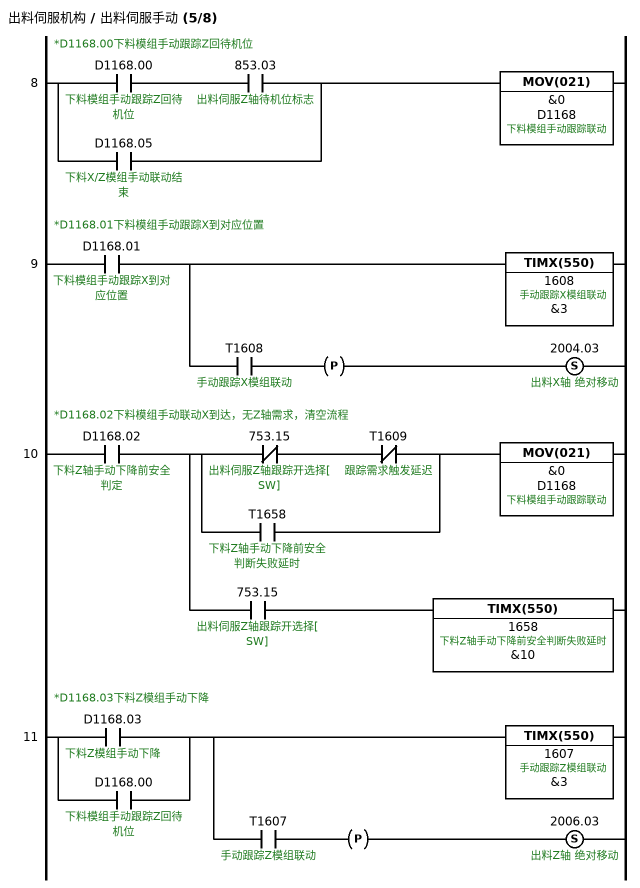
; [picture p480: 出料伺服机构 / 出料伺服手动, rungs 8-11]
; rung 8: *D1168.00下料模组手动跟踪Z回待机位
LD D1168.00  ; 下料模组手动跟踪Z回待机位
AND 853.03  ; 出料伺服Z轴待机位标志
OR D1168.05  ; 下料X/Z模组手动联动结束
MOV(021) &0 D1168  ; 下料模组手动跟踪联动
; rung 9: *D1168.01下料模组手动跟踪X到对应位置
LD D1168.01  ; 下料模组手动跟踪X到对应位置
TIMX(550) 1608 &3  ; 手动跟踪X模组联动
AND T1608  ; 手动跟踪X模组联动
UP(521)
SET 2004.03  ; 出料X轴 绝对移动
; rung 10: *D1168.02下料模组手动联动X到达，无Z轴需求，清空流程
LD D1168.02  ; 下料Z轴手动下降前安全判定
OUT TR0
LDNOT 753.15  ; 出料伺服Z轴跟踪开选择[SW]
ANDNOT T1609  ; 跟踪需求触发延迟
OR T1658  ; 下料Z轴手动下降前安全判断失败延时
ANDLD
MOV(021) &0 D1168  ; 下料模组手动跟踪联动
LD TR0
AND 753.15  ; 出料伺服Z轴跟踪开选择[SW]
TIMX(550) 1658 &10  ; 下料Z轴手动下降前安全判断失败延时
; rung 11: *D1168.03下料Z模组手动下降
LD D1168.03  ; 下料Z模组手动下降
OR D1168.00  ; 下料模组手动跟踪Z回待机位
TIMX(550) 1607 &3  ; 手动跟踪Z模组联动
AND T1607  ; 手动跟踪Z模组联动
UP(521)
SET 2006.03  ; 出料Z轴 绝对移动

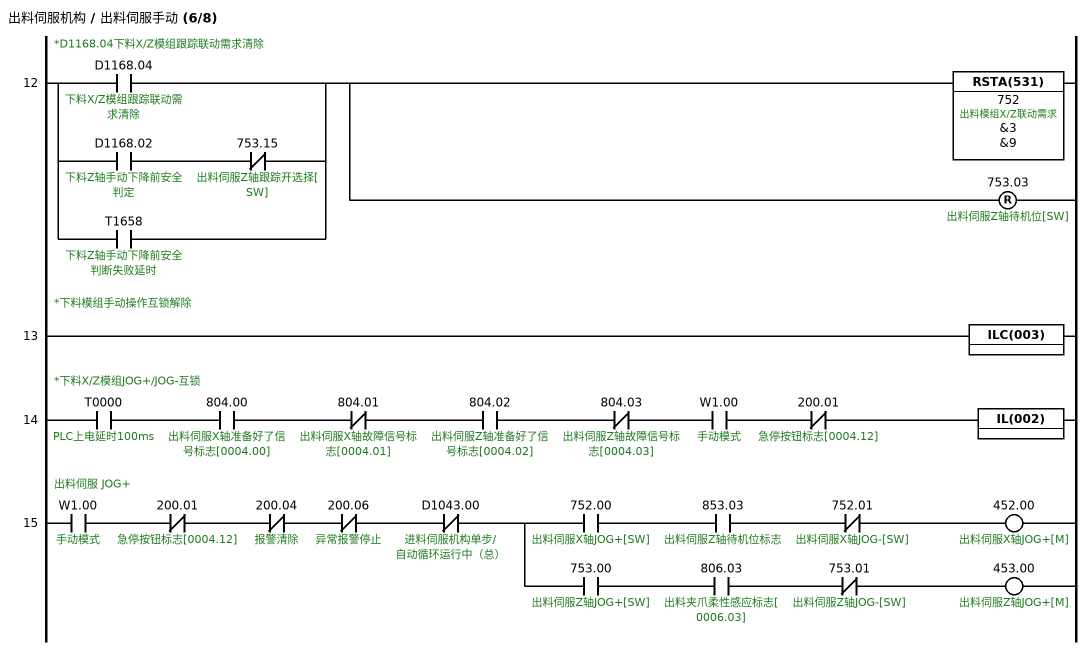
; rung 12: *D1168.04下料X/Z模组跟踪联动需求清除
LD D1168.04  ; 下料X/Z模组跟踪联动需求清除
LD D1168.02  ; 下料Z轴手动下降前安全判定
ANDNOT 753.15  ; 出料伺服Z轴跟踪开选择[SW]
ORLD
OR T1658  ; 下料Z轴手动下降前安全判断失败延时
RSTA(531) 752 &3 &9  ; 出料模组X/Z联动需求
RSET 753.03  ; 出料伺服Z轴待机位[SW]
; rung 13: *下料模组手动操作互锁解除
ILC(003)
; rung 14: *下料X/Z模组JOG+/JOG-互锁
LD T0000  ; PLC上电延时100ms
AND 804.00  ; 出料伺服X轴准备好了信号标志[0004.00]
ANDNOT 804.01  ; 出料伺服X轴故障信号标志[0004.01]
AND 804.02  ; 出料伺服Z轴准备好了信号标志[0004.02]
ANDNOT 804.03  ; 出料伺服Z轴故障信号标志[0004.03]
AND W1.00  ; 手动模式
ANDNOT 200.01  ; 急停按钮标志[0004.12]
IL(002)
; rung 15: 出料伺服 JOG+
LD W1.00  ; 手动模式
ANDNOT 200.01  ; 急停按钮标志[0004.12]
ANDNOT 200.04  ; 报警清除
ANDNOT 200.06  ; 异常报警停止
ANDNOT D1043.00  ; 进料伺服机构单步/自动循环运行中（总）
OUT TR0
AND 752.00  ; 出料伺服X轴JOG+[SW]
AND 853.03  ; 出料伺服Z轴待机位标志
ANDNOT 752.01  ; 出料伺服X轴JOG-[SW]
OUT 452.00  ; 出料伺服X轴JOG+[M]
LD TR0
AND 753.00  ; 出料伺服Z轴JOG+[SW]
AND 806.03  ; 出料夹爪柔性感应标志[0006.03]
ANDNOT 753.01  ; 出料伺服Z轴JOG-[SW]
OUT 453.00  ; 出料伺服Z轴JOG+[M]

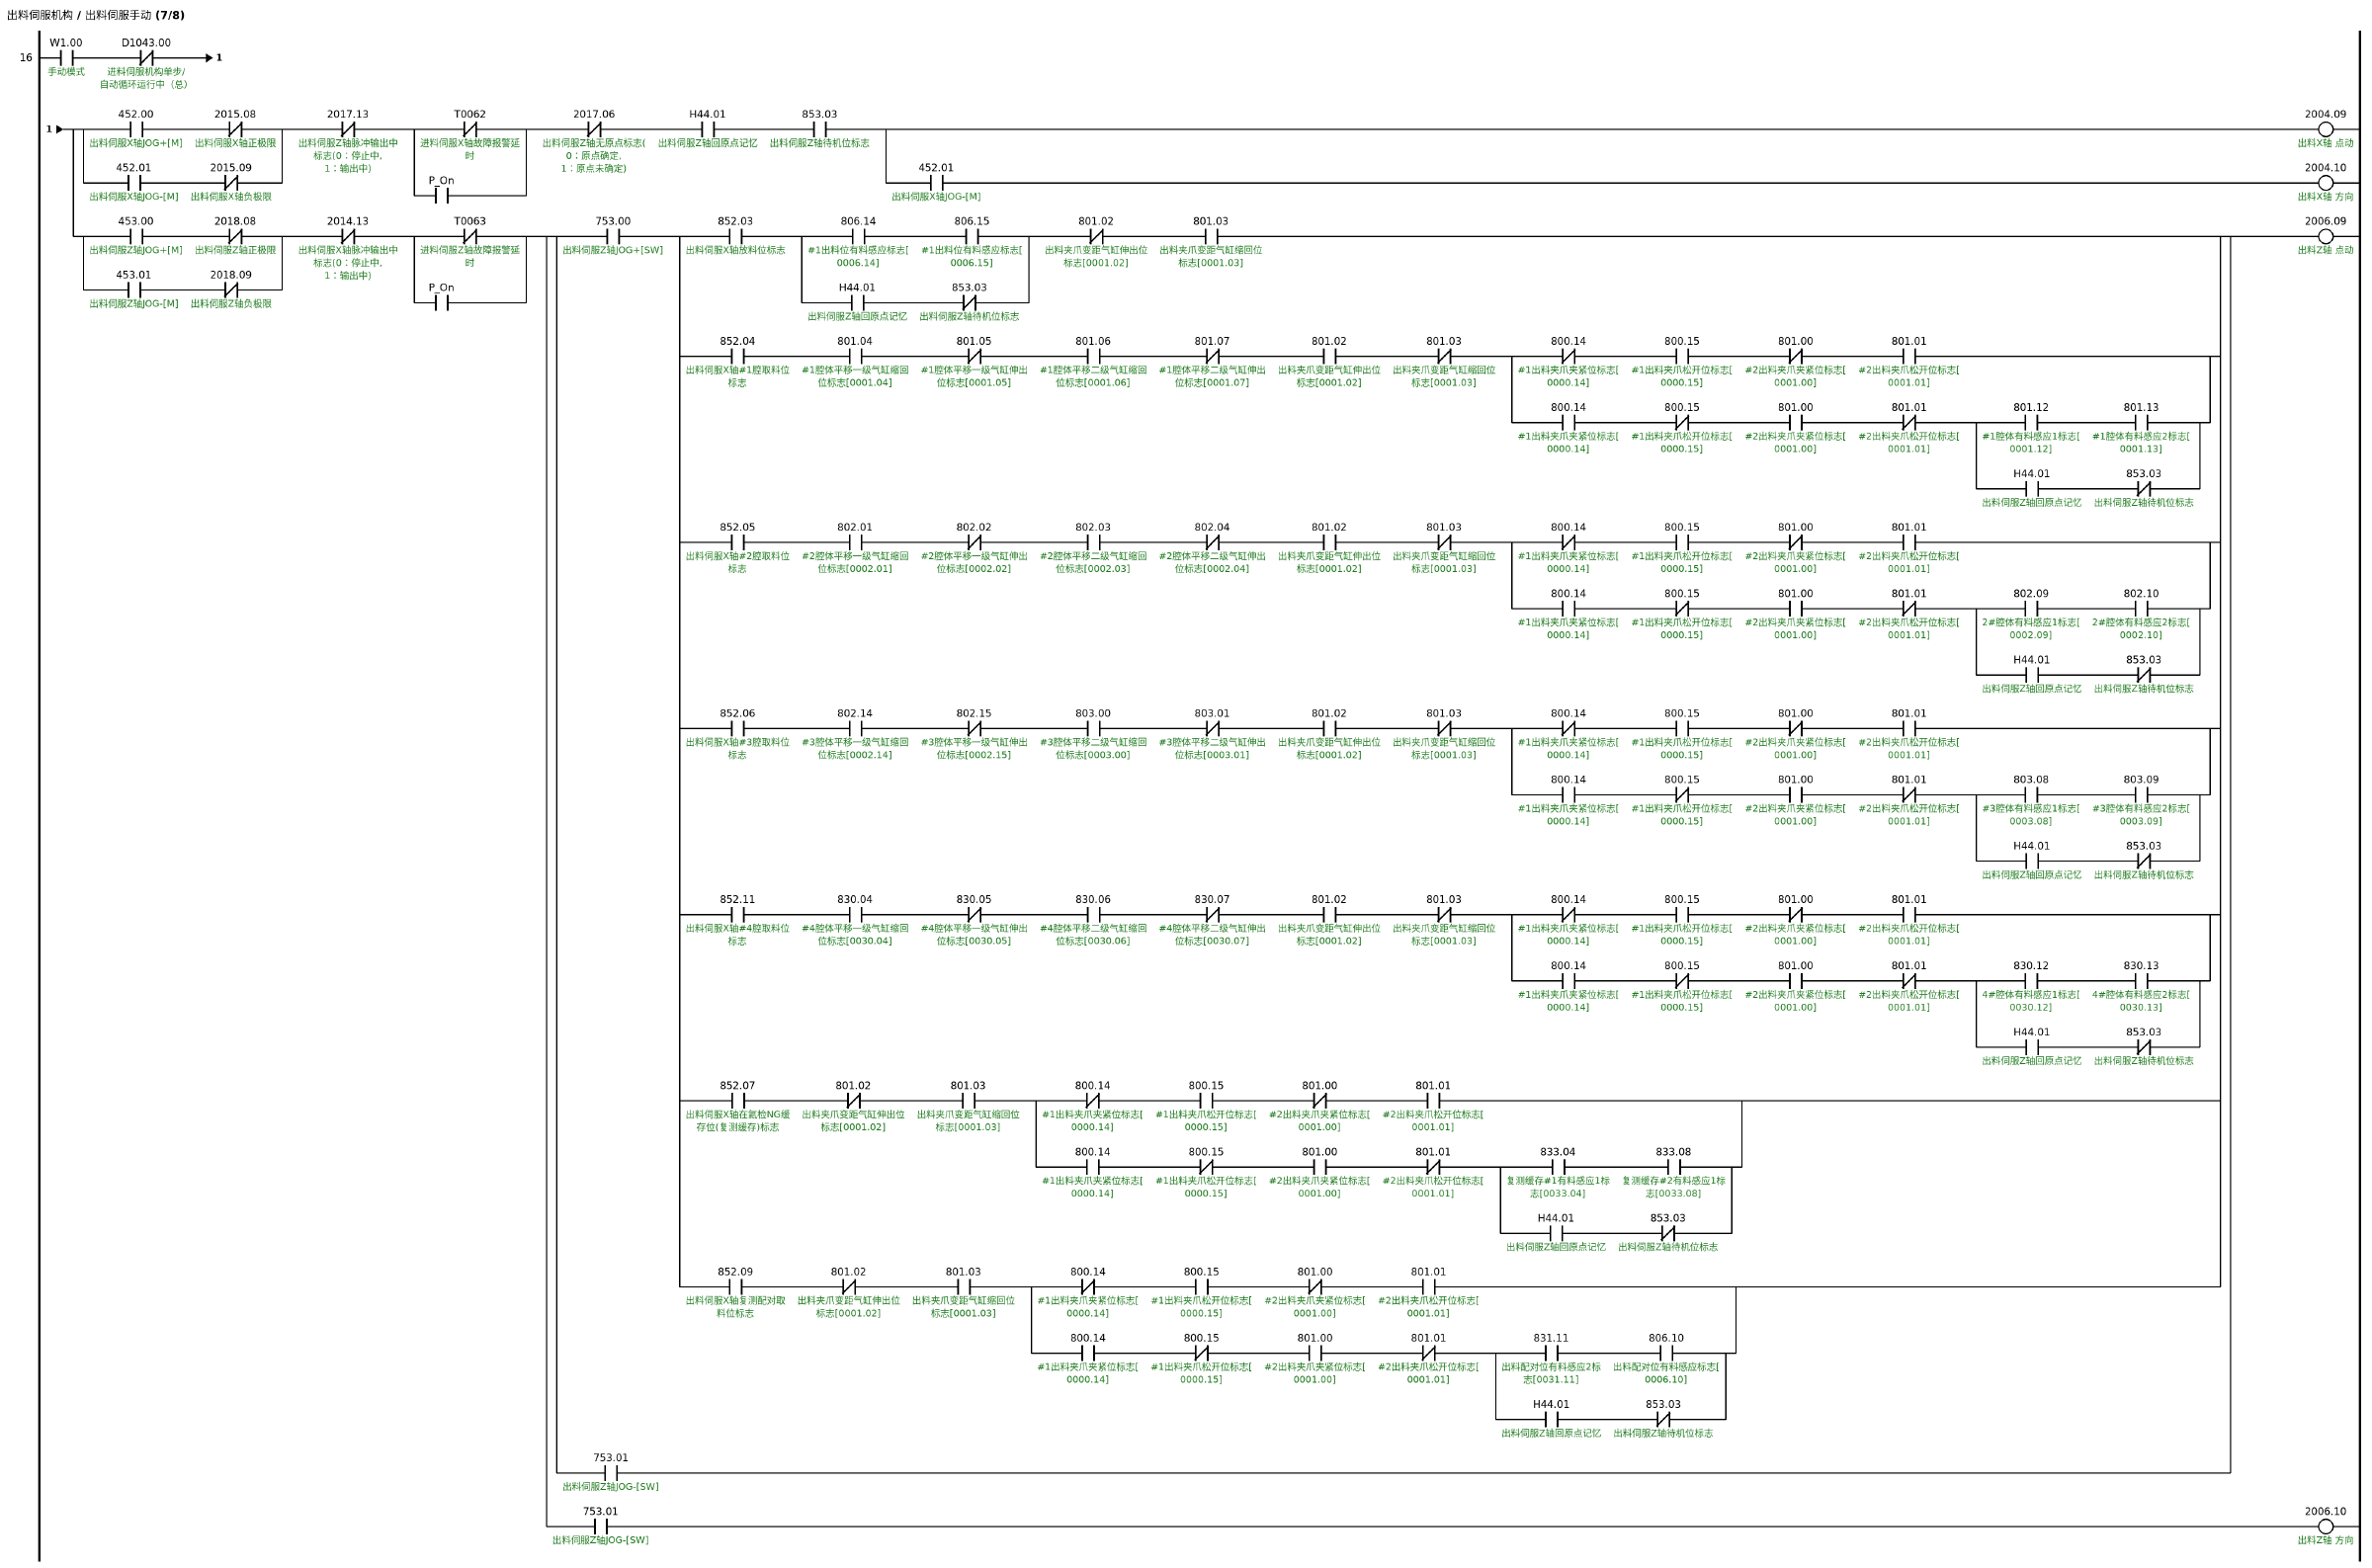
; rung 16
LD W1.00  ; 手动模式
ANDNOT D1043.00  ; 进料伺服机构单步/自动循环运行中（总）
OUT TR0
LD 452.00  ; 出料伺服X轴JOG+[M]
ANDNOT 2015.08  ; 出料伺服X轴正极限
LD 452.01  ; 出料伺服X轴JOG-[M]
ANDNOT 2015.09  ; 出料伺服X轴负极限
ORLD
ANDLD
ANDNOT 2017.13  ; 出料伺服Z轴脉冲输出中标志(0：停止中,1：输出中)
LDNOT T0062  ; 进料伺服X轴故障报警延时
OR P_On
ANDLD
ANDNOT 2017.06  ; 出料伺服Z轴无原点标志(0：原点确定,1：原点未确定)
AND H44.01  ; 出料伺服Z轴回原点记忆
AND 853.03  ; 出料伺服Z轴待机位标志
OUT 2004.09  ; 出料X轴 点动
AND 452.01  ; 出料伺服X轴JOG-[M]
OUT 2004.10  ; 出料X轴 方向
LD TR0
LD 453.00  ; 出料伺服Z轴JOG+[M]
ANDNOT 2018.08  ; 出料伺服Z轴正极限
LD 453.01  ; 出料伺服Z轴JOG-[M]
ANDNOT 2018.09  ; 出料伺服Z轴负极限
ORLD
ANDLD
ANDNOT 2014.13  ; 出料伺服X轴脉冲输出中标志(0：停止中,1：输出中)
LDNOT T0063  ; 进料伺服Z轴故障报警延时
OR P_On
ANDLD
OUT TR0
LD 753.00  ; 出料伺服Z轴JOG+[SW]
LD 852.03  ; 出料伺服X轴放料位标志
LD 806.14  ; #1出料位有料感应标志[0006.14]
AND 806.15  ; #1出料位有料感应标志[0006.15]
LD H44.01  ; 出料伺服Z轴回原点记忆
ANDNOT 853.03  ; 出料伺服Z轴待机位标志
ORLD
ANDLD
ANDNOT 801.02  ; 出料夹爪变距气缸伸出位标志[0001.02]
AND 801.03  ; 出料夹爪变距气缸缩回位标志[0001.03]
LD 852.04  ; 出料伺服X轴#1腔取料位标志
AND 801.04  ; #1腔体平移一级气缸缩回位标志[0001.04]
ANDNOT 801.05  ; #1腔体平移一级气缸伸出位标志[0001.05]
AND 801.06  ; #1腔体平移二级气缸缩回位标志[0001.06]
ANDNOT 801.07  ; #1腔体平移二级气缸伸出位标志[0001.07]
AND 801.02  ; 出料夹爪变距气缸伸出位标志[0001.02]
ANDNOT 801.03  ; 出料夹爪变距气缸缩回位标志[0001.03]
LDNOT 800.14  ; #1出料夹爪夹紧位标志[0000.14]
AND 800.15  ; #1出料夹爪松开位标志[0000.15]
ANDNOT 801.00  ; #2出料夹爪夹紧位标志[0001.00]
AND 801.01  ; #2出料夹爪松开位标志[0001.01]
LD 800.14  ; #1出料夹爪夹紧位标志[0000.14]
ANDNOT 800.15  ; #1出料夹爪松开位标志[0000.15]
AND 801.00  ; #2出料夹爪夹紧位标志[0001.00]
ANDNOT 801.01  ; #2出料夹爪松开位标志[0001.01]
LD 801.12  ; #1腔体有料感应1标志[0001.12]
AND 801.13  ; #1腔体有料感应2标志[0001.13]
LD H44.01  ; 出料伺服Z轴回原点记忆
ANDNOT 853.03  ; 出料伺服Z轴待机位标志
ORLD
ANDLD
ORLD
ANDLD
ORLD
LD 852.05  ; 出料伺服X轴#2腔取料位标志
AND 802.01  ; #2腔体平移一级气缸缩回位标志[0002.01]
ANDNOT 802.02  ; #2腔体平移一级气缸伸出位标志[0002.02]
AND 802.03  ; #2腔体平移二级气缸缩回位标志[0002.03]
ANDNOT 802.04  ; #2腔体平移二级气缸伸出位标志[0002.04]
AND 801.02  ; 出料夹爪变距气缸伸出位标志[0001.02]
ANDNOT 801.03  ; 出料夹爪变距气缸缩回位标志[0001.03]
LDNOT 800.14  ; #1出料夹爪夹紧位标志[0000.14]
AND 800.15  ; #1出料夹爪松开位标志[0000.15]
ANDNOT 801.00  ; #2出料夹爪夹紧位标志[0001.00]
AND 801.01  ; #2出料夹爪松开位标志[0001.01]
LD 800.14  ; #1出料夹爪夹紧位标志[0000.14]
ANDNOT 800.15  ; #1出料夹爪松开位标志[0000.15]
AND 801.00  ; #2出料夹爪夹紧位标志[0001.00]
ANDNOT 801.01  ; #2出料夹爪松开位标志[0001.01]
LD 802.09  ; 2#腔体有料感应1标志[0002.09]
AND 802.10  ; 2#腔体有料感应2标志[0002.10]
LD H44.01  ; 出料伺服Z轴回原点记忆
ANDNOT 853.03  ; 出料伺服Z轴待机位标志
ORLD
ANDLD
ORLD
ANDLD
ORLD
LD 852.06  ; 出料伺服X轴#3腔取料位标志
AND 802.14  ; #3腔体平移一级气缸缩回位标志[0002.14]
ANDNOT 802.15  ; #3腔体平移一级气缸伸出位标志[0002.15]
AND 803.00  ; #3腔体平移二级气缸缩回位标志[0003.00]
ANDNOT 803.01  ; #3腔体平移二级气缸伸出位标志[0003.01]
AND 801.02  ; 出料夹爪变距气缸伸出位标志[0001.02]
ANDNOT 801.03  ; 出料夹爪变距气缸缩回位标志[0001.03]
LDNOT 800.14  ; #1出料夹爪夹紧位标志[0000.14]
AND 800.15  ; #1出料夹爪松开位标志[0000.15]
ANDNOT 801.00  ; #2出料夹爪夹紧位标志[0001.00]
AND 801.01  ; #2出料夹爪松开位标志[0001.01]
LD 800.14  ; #1出料夹爪夹紧位标志[0000.14]
ANDNOT 800.15  ; #1出料夹爪松开位标志[0000.15]
AND 801.00  ; #2出料夹爪夹紧位标志[0001.00]
ANDNOT 801.01  ; #2出料夹爪松开位标志[0001.01]
LD 803.08  ; #3腔体有料感应1标志[0003.08]
AND 803.09  ; #3腔体有料感应2标志[0003.09]
LD H44.01  ; 出料伺服Z轴回原点记忆
ANDNOT 853.03  ; 出料伺服Z轴待机位标志
ORLD
ANDLD
ORLD
ANDLD
ORLD
LD 852.11  ; 出料伺服X轴#4腔取料位标志
AND 830.04  ; #4腔体平移一级气缸缩回位标志[0030.04]
ANDNOT 830.05  ; #4腔体平移一级气缸伸出位标志[0030.05]
AND 830.06  ; #4腔体平移二级气缸缩回位标志[0030.06]
ANDNOT 830.07  ; #4腔体平移二级气缸伸出位标志[0030.07]
AND 801.02  ; 出料夹爪变距气缸伸出位标志[0001.02]
ANDNOT 801.03  ; 出料夹爪变距气缸缩回位标志[0001.03]
LDNOT 800.14  ; #1出料夹爪夹紧位标志[0000.14]
AND 800.15  ; #1出料夹爪松开位标志[0000.15]
ANDNOT 801.00  ; #2出料夹爪夹紧位标志[0001.00]
AND 801.01  ; #2出料夹爪松开位标志[0001.01]
LD 800.14  ; #1出料夹爪夹紧位标志[0000.14]
ANDNOT 800.15  ; #1出料夹爪松开位标志[0000.15]
AND 801.00  ; #2出料夹爪夹紧位标志[0001.00]
ANDNOT 801.01  ; #2出料夹爪松开位标志[0001.01]
LD 830.12  ; 4#腔体有料感应1标志[0030.12]
AND 830.13  ; 4#腔体有料感应2标志[0030.13]
LD H44.01  ; 出料伺服Z轴回原点记忆
ANDNOT 853.03  ; 出料伺服Z轴待机位标志
ORLD
ANDLD
ORLD
ANDLD
ORLD
LD 852.07  ; 出料伺服X轴在氦检NG缓存位(复测缓存)标志
ANDNOT 801.02  ; 出料夹爪变距气缸伸出位标志[0001.02]
AND 801.03  ; 出料夹爪变距气缸缩回位标志[0001.03]
LDNOT 800.14  ; #1出料夹爪夹紧位标志[0000.14]
AND 800.15  ; #1出料夹爪松开位标志[0000.15]
ANDNOT 801.00  ; #2出料夹爪夹紧位标志[0001.00]
AND 801.01  ; #2出料夹爪松开位标志[0001.01]
LD 800.14  ; #1出料夹爪夹紧位标志[0000.14]
ANDNOT 800.15  ; #1出料夹爪松开位标志[0000.15]
AND 801.00  ; #2出料夹爪夹紧位标志[0001.00]
ANDNOT 801.01  ; #2出料夹爪松开位标志[0001.01]
LD 833.04  ; 复测缓存#1有料感应1标志[0033.04]
AND 833.08  ; 复测缓存#2有料感应1标志[0033.08]
LD H44.01  ; 出料伺服Z轴回原点记忆
ANDNOT 853.03  ; 出料伺服Z轴待机位标志
ORLD
ANDLD
ORLD
ANDLD
ORLD
LD 852.09  ; 出料伺服X轴复测配对取料位标志
ANDNOT 801.02  ; 出料夹爪变距气缸伸出位标志[0001.02]
AND 801.03  ; 出料夹爪变距气缸缩回位标志[0001.03]
LDNOT 800.14  ; #1出料夹爪夹紧位标志[0000.14]
AND 800.15  ; #1出料夹爪松开位标志[0000.15]
ANDNOT 801.00  ; #2出料夹爪夹紧位标志[0001.00]
AND 801.01  ; #2出料夹爪松开位标志[0001.01]
LD 800.14  ; #1出料夹爪夹紧位标志[0000.14]
ANDNOT 800.15  ; #1出料夹爪松开位标志[0000.15]
AND 801.00  ; #2出料夹爪夹紧位标志[0001.00]
ANDNOT 801.01  ; #2出料夹爪松开位标志[0001.01]
LD 831.11  ; 出料配对位有料感应2标志[0031.11]
AND 806.10  ; 出料配对位有料感应标志[0006.10]
LD H44.01  ; 出料伺服Z轴回原点记忆
ANDNOT 853.03  ; 出料伺服Z轴待机位标志
ORLD
ANDLD
ORLD
ANDLD
ORLD
ANDLD
OR 753.01  ; 出料伺服Z轴JOG-[SW]
ANDLD
OUT 2006.09  ; 出料Z轴 点动
LD TR0
AND 753.01  ; 出料伺服Z轴JOG-[SW]
OUT 2006.10  ; 出料Z轴 方向

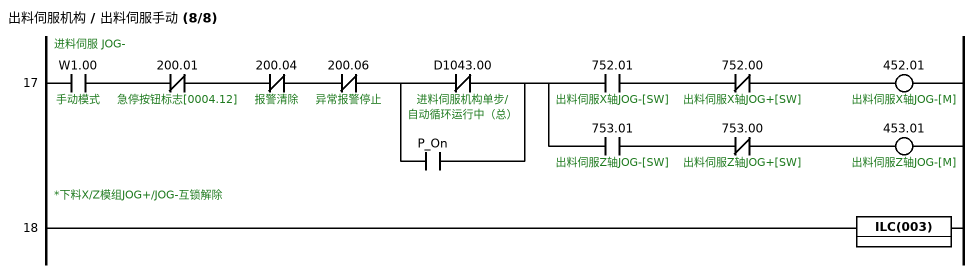
; rung 17: 进料伺服 JOG-
LD W1.00  ; 手动模式
ANDNOT 200.01  ; 急停按钮标志[0004.12]
ANDNOT 200.04  ; 报警清除
ANDNOT 200.06  ; 异常报警停止
LDNOT D1043.00  ; 进料伺服机构单步/自动循环运行中（总）
OR P_On
ANDLD
OUT TR0
AND 752.01  ; 出料伺服X轴JOG-[SW]
ANDNOT 752.00  ; 出料伺服X轴JOG+[SW]
OUT 452.01  ; 出料伺服X轴JOG-[M]
LD TR0
AND 753.01  ; 出料伺服Z轴JOG-[SW]
ANDNOT 753.00  ; 出料伺服Z轴JOG+[SW]
OUT 453.01  ; 出料伺服Z轴JOG-[M]
; rung 18: *下料X/Z模组JOG+/JOG-互锁解除
ILC(003)

### Section 出料伺服自动

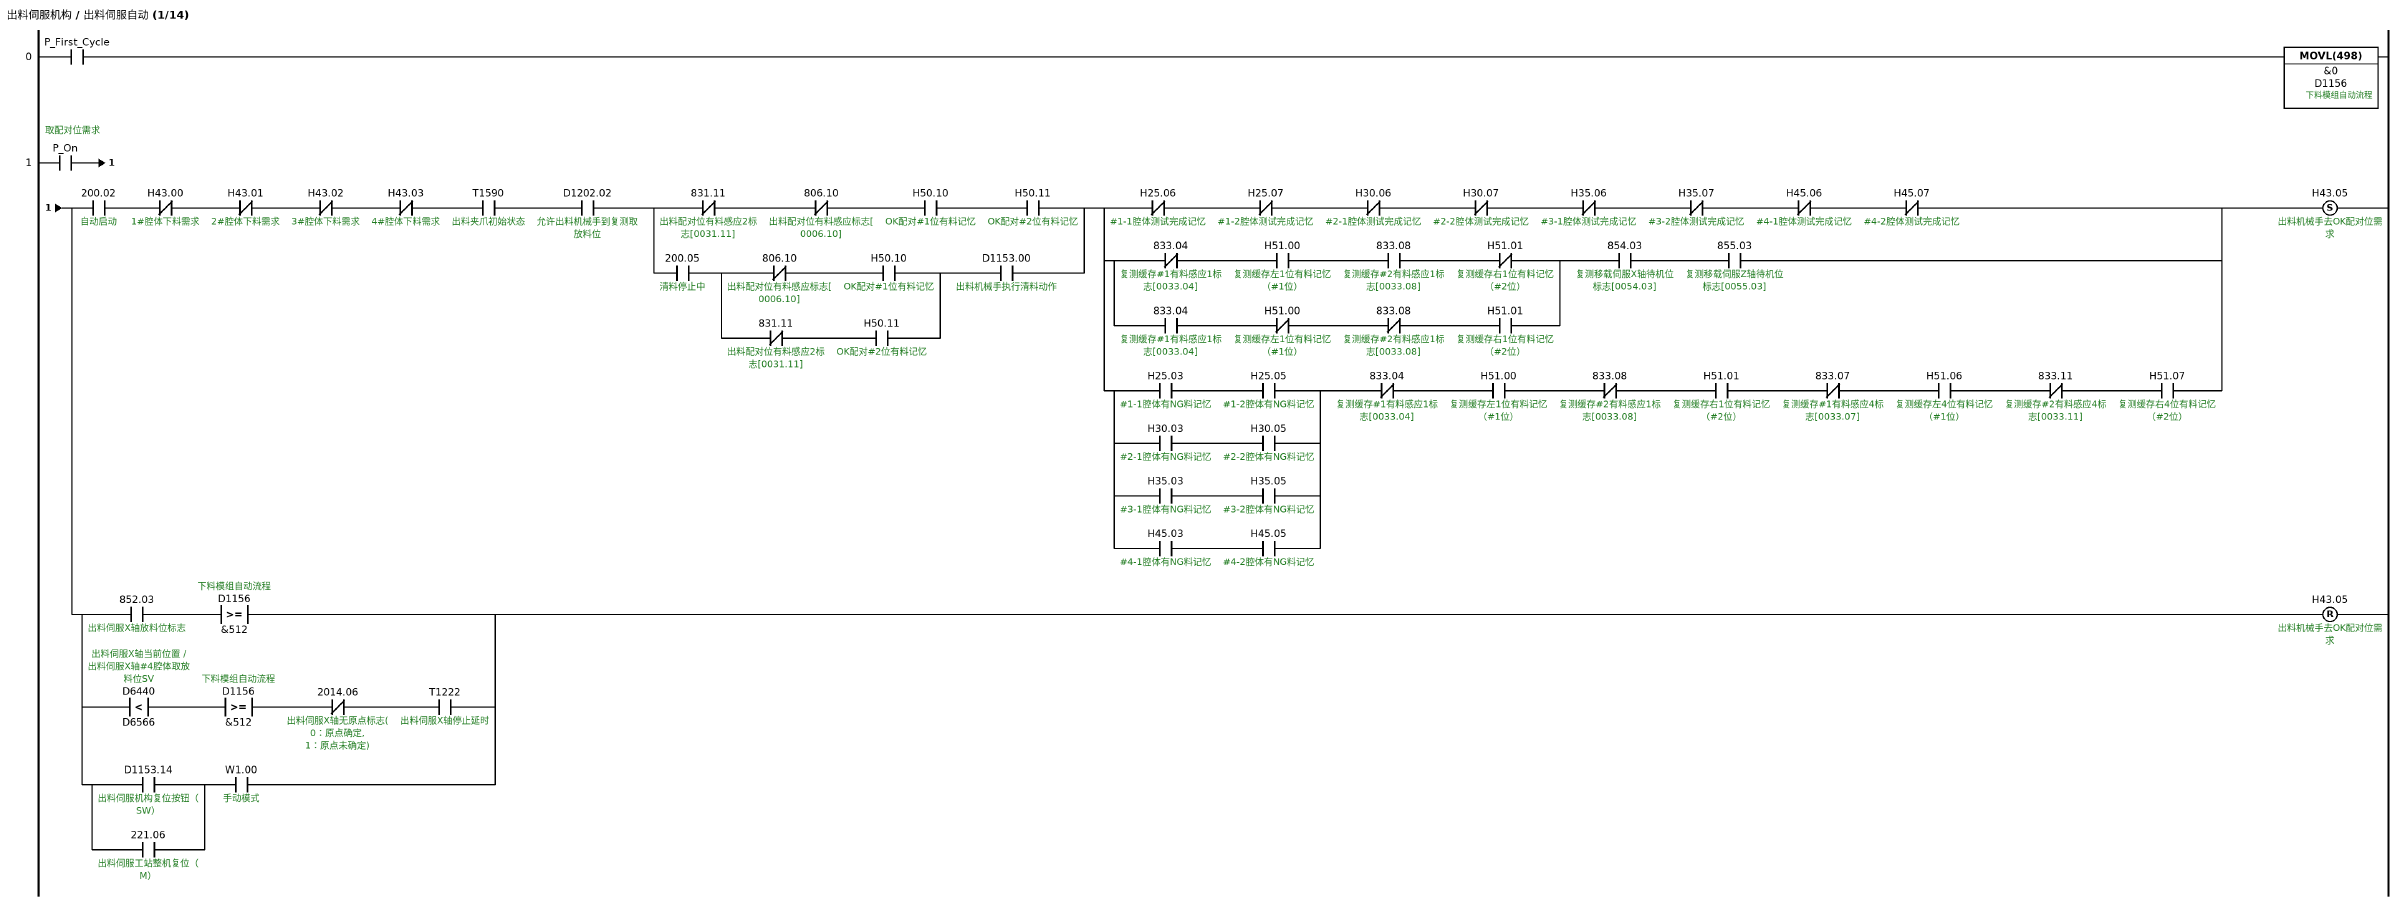
; rung 0
LD P_First_Cycle
MOVL(498) &0 D1156  ; 下料模组自动流程
; rung 1: 取配对位需求
LD P_On
OUT TR0
AND 200.02  ; 自动启动
ANDNOT H43.00  ; 1#腔体下料需求
ANDNOT H43.01  ; 2#腔体下料需求
ANDNOT H43.02  ; 3#腔体下料需求
ANDNOT H43.03  ; 4#腔体下料需求
AND T1590  ; 出料夹爪初始状态
AND D1202.02  ; 允许出料机械手到复测取放料位
LDNOT 831.11  ; 出料配对位有料感应2标志[0031.11]
ANDNOT 806.10  ; 出料配对位有料感应标志[0006.10]
AND H50.10  ; OK配对#1位有料记忆
AND H50.11  ; OK配对#2位有料记忆
LD 200.05  ; 清料停止中
LDNOT 806.10  ; 出料配对位有料感应标志[0006.10]
AND H50.10  ; OK配对#1位有料记忆
LDNOT 831.11  ; 出料配对位有料感应2标志[0031.11]
AND H50.11  ; OK配对#2位有料记忆
ORLD
ANDLD
AND D1153.00  ; 出料机械手执行清料动作
ORLD
ANDLD
LDNOT H25.06  ; #1-1腔体测试完成记忆
ANDNOT H25.07  ; #1-2腔体测试完成记忆
ANDNOT H30.06  ; #2-1腔体测试完成记忆
ANDNOT H30.07  ; #2-2腔体测试完成记忆
ANDNOT H35.06  ; #3-1腔体测试完成记忆
ANDNOT H35.07  ; #3-2腔体测试完成记忆
ANDNOT H45.06  ; #4-1腔体测试完成记忆
ANDNOT H45.07  ; #4-2腔体测试完成记忆
LDNOT 833.04  ; 复测缓存#1有料感应1标志[0033.04]
AND H51.00  ; 复测缓存左1位有料记忆（#1位）
AND 833.08  ; 复测缓存#2有料感应1标志[0033.08]
ANDNOT H51.01  ; 复测缓存右1位有料记忆（#2位）
LD 833.04  ; 复测缓存#1有料感应1标志[0033.04]
ANDNOT H51.00  ; 复测缓存左1位有料记忆（#1位）
ANDNOT 833.08  ; 复测缓存#2有料感应1标志[0033.08]
AND H51.01  ; 复测缓存右1位有料记忆（#2位）
ORLD
AND 854.03  ; 复测移载伺服X轴待机位标志[0054.03]
AND 855.03  ; 复测移载伺服Z轴待机位标志[0055.03]
ORLD
LD H25.03  ; #1-1腔体有NG料记忆
AND H25.05  ; #1-2腔体有NG料记忆
LD H30.03  ; #2-1腔体有NG料记忆
AND H30.05  ; #2-2腔体有NG料记忆
ORLD
LD H35.03  ; #3-1腔体有NG料记忆
AND H35.05  ; #3-2腔体有NG料记忆
ORLD
LD H45.03  ; #4-1腔体有NG料记忆
AND H45.05  ; #4-2腔体有NG料记忆
ORLD
ANDNOT 833.04  ; 复测缓存#1有料感应1标志[0033.04]
AND H51.00  ; 复测缓存左1位有料记忆（#1位）
ANDNOT 833.08  ; 复测缓存#2有料感应1标志[0033.08]
AND H51.01  ; 复测缓存右1位有料记忆（#2位）
ANDNOT 833.07  ; 复测缓存#1有料感应4标志[0033.07]
AND H51.06  ; 复测缓存左4位有料记忆（#1位）
ANDNOT 833.11  ; 复测缓存#2有料感应4标志[0033.11]
AND H51.07  ; 复测缓存右4位有料记忆（#2位）
ORLD
ANDLD
SET H43.05  ; 出料机械手去OK配对位需求
LD TR0
LD 852.03  ; 出料伺服X轴放料位标志
AND>=(325) D1156 &512  ; 下料模组自动流程
LD<SL(313) D6440 D6566  ; 出料伺服X轴当前位置, 出料伺服X轴#4腔体取放料位SV
AND>=(325) D1156 &512  ; 下料模组自动流程
ANDNOT 2014.06  ; 出料伺服X轴无原点标志(0：原点确定,1：原点未确定)
AND T1222  ; 出料伺服X轴停止延时
ORLD
LD D1153.14  ; 出料伺服机构复位按钮（SW）
OR 221.06  ; 出料伺服工站整机复位（M）
AND W1.00  ; 手动模式
ORLD
ANDLD
RSET H43.05  ; 出料机械手去OK配对位需求

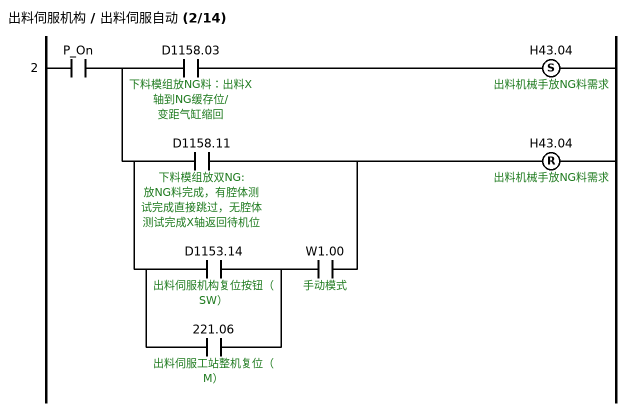
; rung 2
LD P_On
OUT TR0
AND D1158.03  ; 下料模组放NG料：出料X轴到NG缓存位/变距气缸缩回
SET H43.04  ; 出料机械手放NG料需求
LD TR0
LD D1158.11  ; 下料模组放双NG:放NG料完成，有腔体测试完成直接跳过，无腔体测试完成X轴返回待机位
LD D1153.14  ; 出料伺服机构复位按钮（SW）
OR 221.06  ; 出料伺服工站整机复位（M）
AND W1.00  ; 手动模式
ORLD
ANDLD
RSET H43.04  ; 出料机械手放NG料需求

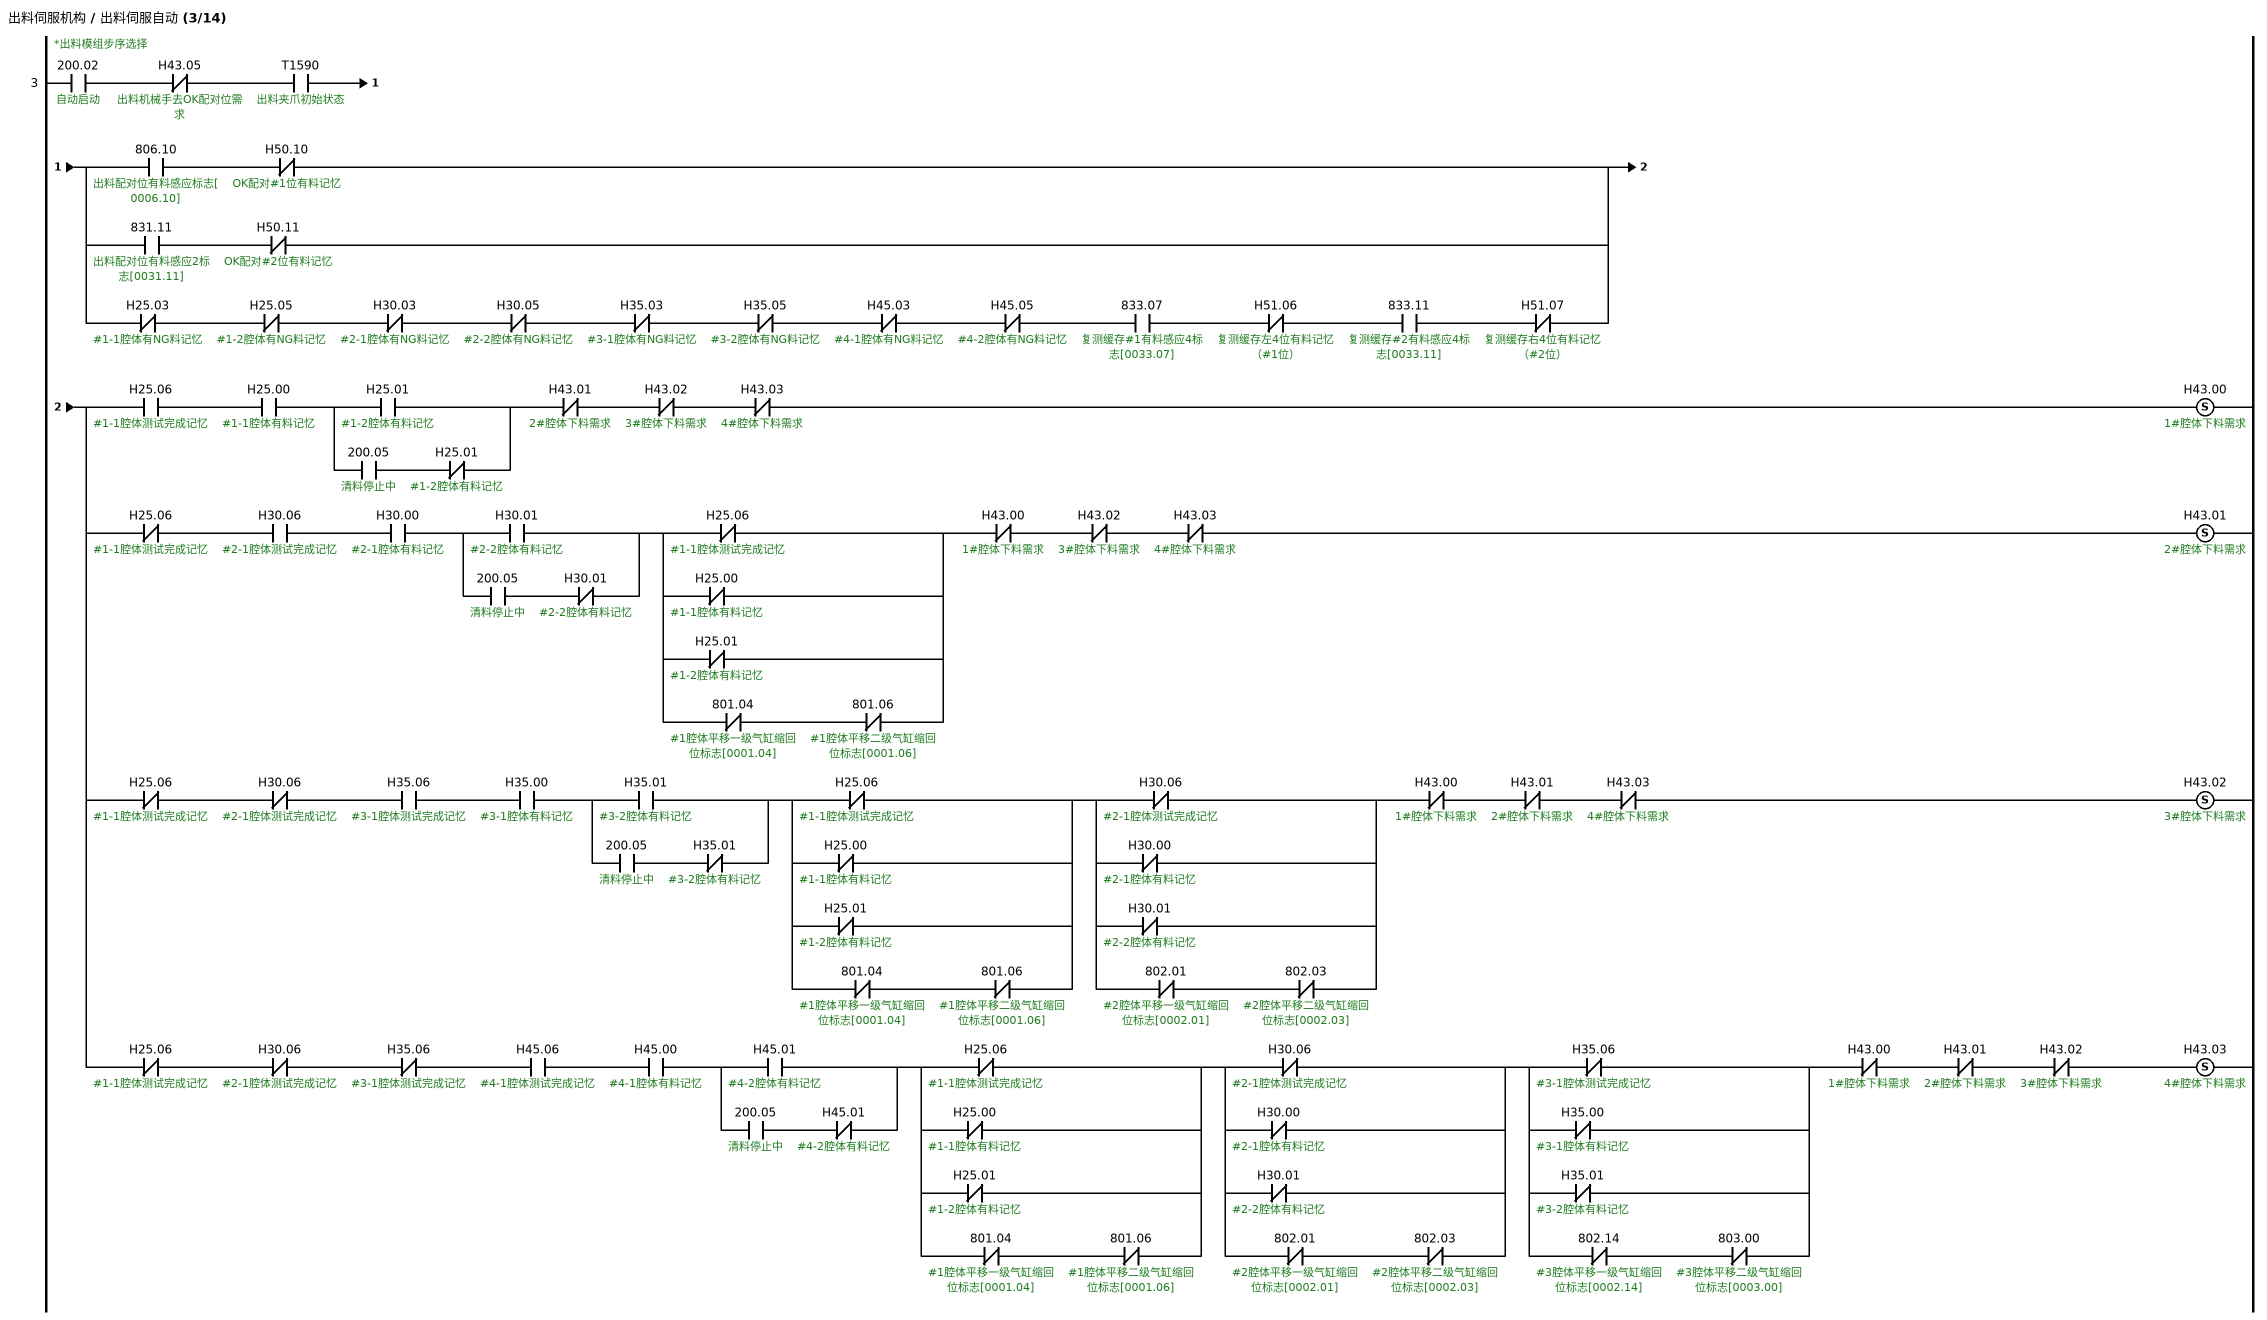
; rung 3: *出料模组步序选择
LD 200.02  ; 自动启动
ANDNOT H43.05  ; 出料机械手去OK配对位需求
AND T1590  ; 出料夹爪初始状态
LD 806.10  ; 出料配对位有料感应标志[0006.10]
ANDNOT H50.10  ; OK配对#1位有料记忆
LD 831.11  ; 出料配对位有料感应2标志[0031.11]
ANDNOT H50.11  ; OK配对#2位有料记忆
ORLD
LDNOT H25.03  ; #1-1腔体有NG料记忆
ANDNOT H25.05  ; #1-2腔体有NG料记忆
ANDNOT H30.03  ; #2-1腔体有NG料记忆
ANDNOT H30.05  ; #2-2腔体有NG料记忆
ANDNOT H35.03  ; #3-1腔体有NG料记忆
ANDNOT H35.05  ; #3-2腔体有NG料记忆
ANDNOT H45.03  ; #4-1腔体有NG料记忆
ANDNOT H45.05  ; #4-2腔体有NG料记忆
AND 833.07  ; 复测缓存#1有料感应4标志[0033.07]
ANDNOT H51.06  ; 复测缓存左4位有料记忆（#1位）
AND 833.11  ; 复测缓存#2有料感应4标志[0033.11]
ANDNOT H51.07  ; 复测缓存右4位有料记忆（#2位）
ORLD
ANDLD
OUT TR0
AND H25.06  ; #1-1腔体测试完成记忆
AND H25.00  ; #1-1腔体有料记忆
LD H25.01  ; #1-2腔体有料记忆
LD 200.05  ; 清料停止中
ANDNOT H25.01  ; #1-2腔体有料记忆
ORLD
ANDLD
ANDNOT H43.01  ; 2#腔体下料需求
ANDNOT H43.02  ; 3#腔体下料需求
ANDNOT H43.03  ; 4#腔体下料需求
SET H43.00  ; 1#腔体下料需求
LD TR0
ANDNOT H25.06  ; #1-1腔体测试完成记忆
AND H30.06  ; #2-1腔体测试完成记忆
AND H30.00  ; #2-1腔体有料记忆
LD H30.01  ; #2-2腔体有料记忆
LD 200.05  ; 清料停止中
ANDNOT H30.01  ; #2-2腔体有料记忆
ORLD
ANDLD
LDNOT H25.06  ; #1-1腔体测试完成记忆
ORNOT H25.00  ; #1-1腔体有料记忆
ORNOT H25.01  ; #1-2腔体有料记忆
LDNOT 801.04  ; #1腔体平移一级气缸缩回位标志[0001.04]
ANDNOT 801.06  ; #1腔体平移二级气缸缩回位标志[0001.06]
ORLD
ANDLD
ANDNOT H43.00  ; 1#腔体下料需求
ANDNOT H43.02  ; 3#腔体下料需求
ANDNOT H43.03  ; 4#腔体下料需求
SET H43.01  ; 2#腔体下料需求
LD TR0
ANDNOT H25.06  ; #1-1腔体测试完成记忆
ANDNOT H30.06  ; #2-1腔体测试完成记忆
AND H35.06  ; #3-1腔体测试完成记忆
AND H35.00  ; #3-1腔体有料记忆
LD H35.01  ; #3-2腔体有料记忆
LD 200.05  ; 清料停止中
ANDNOT H35.01  ; #3-2腔体有料记忆
ORLD
ANDLD
LDNOT H25.06  ; #1-1腔体测试完成记忆
ORNOT H25.00  ; #1-1腔体有料记忆
ORNOT H25.01  ; #1-2腔体有料记忆
LDNOT 801.04  ; #1腔体平移一级气缸缩回位标志[0001.04]
ANDNOT 801.06  ; #1腔体平移二级气缸缩回位标志[0001.06]
ORLD
ANDLD
LDNOT H30.06  ; #2-1腔体测试完成记忆
ORNOT H30.00  ; #2-1腔体有料记忆
ORNOT H30.01  ; #2-2腔体有料记忆
LDNOT 802.01  ; #2腔体平移一级气缸缩回位标志[0002.01]
ANDNOT 802.03  ; #2腔体平移二级气缸缩回位标志[0002.03]
ORLD
ANDLD
ANDNOT H43.00  ; 1#腔体下料需求
ANDNOT H43.01  ; 2#腔体下料需求
ANDNOT H43.03  ; 4#腔体下料需求
SET H43.02  ; 3#腔体下料需求
LD TR0
ANDNOT H25.06  ; #1-1腔体测试完成记忆
ANDNOT H30.06  ; #2-1腔体测试完成记忆
ANDNOT H35.06  ; #3-1腔体测试完成记忆
AND H45.06  ; #4-1腔体测试完成记忆
AND H45.00  ; #4-1腔体有料记忆
LD H45.01  ; #4-2腔体有料记忆
LD 200.05  ; 清料停止中
ANDNOT H45.01  ; #4-2腔体有料记忆
ORLD
ANDLD
LDNOT H25.06  ; #1-1腔体测试完成记忆
ORNOT H25.00  ; #1-1腔体有料记忆
ORNOT H25.01  ; #1-2腔体有料记忆
LDNOT 801.04  ; #1腔体平移一级气缸缩回位标志[0001.04]
ANDNOT 801.06  ; #1腔体平移二级气缸缩回位标志[0001.06]
ORLD
ANDLD
LDNOT H30.06  ; #2-1腔体测试完成记忆
ORNOT H30.00  ; #2-1腔体有料记忆
ORNOT H30.01  ; #2-2腔体有料记忆
LDNOT 802.01  ; #2腔体平移一级气缸缩回位标志[0002.01]
ANDNOT 802.03  ; #2腔体平移二级气缸缩回位标志[0002.03]
ORLD
ANDLD
LDNOT H35.06  ; #3-1腔体测试完成记忆
ORNOT H35.00  ; #3-1腔体有料记忆
ORNOT H35.01  ; #3-2腔体有料记忆
LDNOT 802.14  ; #3腔体平移一级气缸缩回位标志[0002.14]
ANDNOT 803.00  ; #3腔体平移二级气缸缩回位标志[0003.00]
ORLD
ANDLD
ANDNOT H43.00  ; 1#腔体下料需求
ANDNOT H43.01  ; 2#腔体下料需求
ANDNOT H43.02  ; 3#腔体下料需求
SET H43.03  ; 4#腔体下料需求

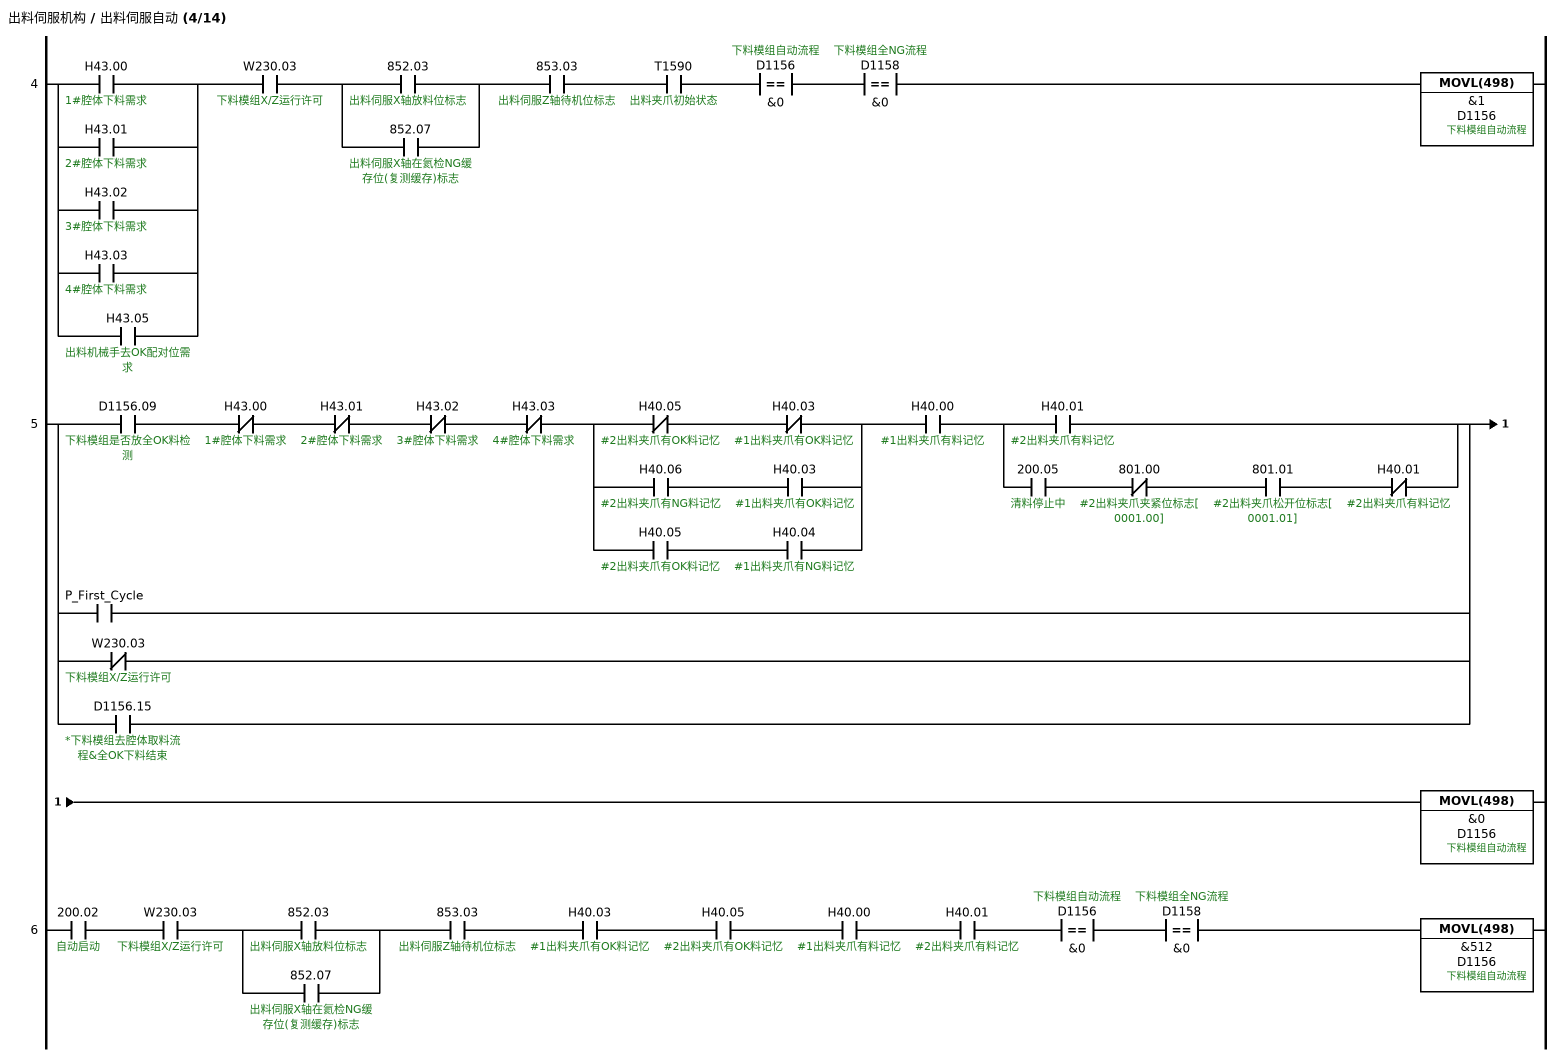
; rung 4
LD H43.00  ; 1#腔体下料需求
OR H43.01  ; 2#腔体下料需求
OR H43.02  ; 3#腔体下料需求
OR H43.03  ; 4#腔体下料需求
OR H43.05  ; 出料机械手去OK配对位需求
AND W230.03  ; 下料模组X/Z运行许可
LD 852.03  ; 出料伺服X轴放料位标志
OR 852.07  ; 出料伺服X轴在氦检NG缓存位(复测缓存)标志
ANDLD
AND 853.03  ; 出料伺服Z轴待机位标志
AND T1590  ; 出料夹爪初始状态
AND=L(301) D1156 &0  ; 下料模组自动流程
AND=L(301) D1158 &0  ; 下料模组全NG流程
MOVL(498) &1 D1156  ; 下料模组自动流程
; rung 5
LD D1156.09  ; 下料模组是否放全OK料检测
ANDNOT H43.00  ; 1#腔体下料需求
ANDNOT H43.01  ; 2#腔体下料需求
ANDNOT H43.02  ; 3#腔体下料需求
ANDNOT H43.03  ; 4#腔体下料需求
LDNOT H40.05  ; #2出料夹爪有OK料记忆
ANDNOT H40.03  ; #1出料夹爪有OK料记忆
LD H40.06  ; #2出料夹爪有NG料记忆
AND H40.03  ; #1出料夹爪有OK料记忆
ORLD
LD H40.05  ; #2出料夹爪有OK料记忆
AND H40.04  ; #1出料夹爪有NG料记忆
ORLD
ANDLD
AND H40.00  ; #1出料夹爪有料记忆
LD H40.01  ; #2出料夹爪有料记忆
LD 200.05  ; 清料停止中
ANDNOT 801.00  ; #2出料夹爪夹紧位标志[0001.00]
AND 801.01  ; #2出料夹爪松开位标志[0001.01]
ANDNOT H40.01  ; #2出料夹爪有料记忆
ORLD
ANDLD
OR P_First_Cycle
ORNOT W230.03  ; 下料模组X/Z运行许可
OR D1156.15  ; *下料模组去腔体取料流程&全OK下料结束
MOVL(498) &0 D1156  ; 下料模组自动流程
; rung 6
LD 200.02  ; 自动启动
AND W230.03  ; 下料模组X/Z运行许可
LD 852.03  ; 出料伺服X轴放料位标志
OR 852.07  ; 出料伺服X轴在氦检NG缓存位(复测缓存)标志
ANDLD
AND 853.03  ; 出料伺服Z轴待机位标志
AND H40.03  ; #1出料夹爪有OK料记忆
AND H40.05  ; #2出料夹爪有OK料记忆
AND H40.00  ; #1出料夹爪有料记忆
AND H40.01  ; #2出料夹爪有料记忆
AND=L(301) D1156 &0  ; 下料模组自动流程
AND=L(301) D1158 &0  ; 下料模组全NG流程
MOVL(498) &512 D1156  ; 下料模组自动流程

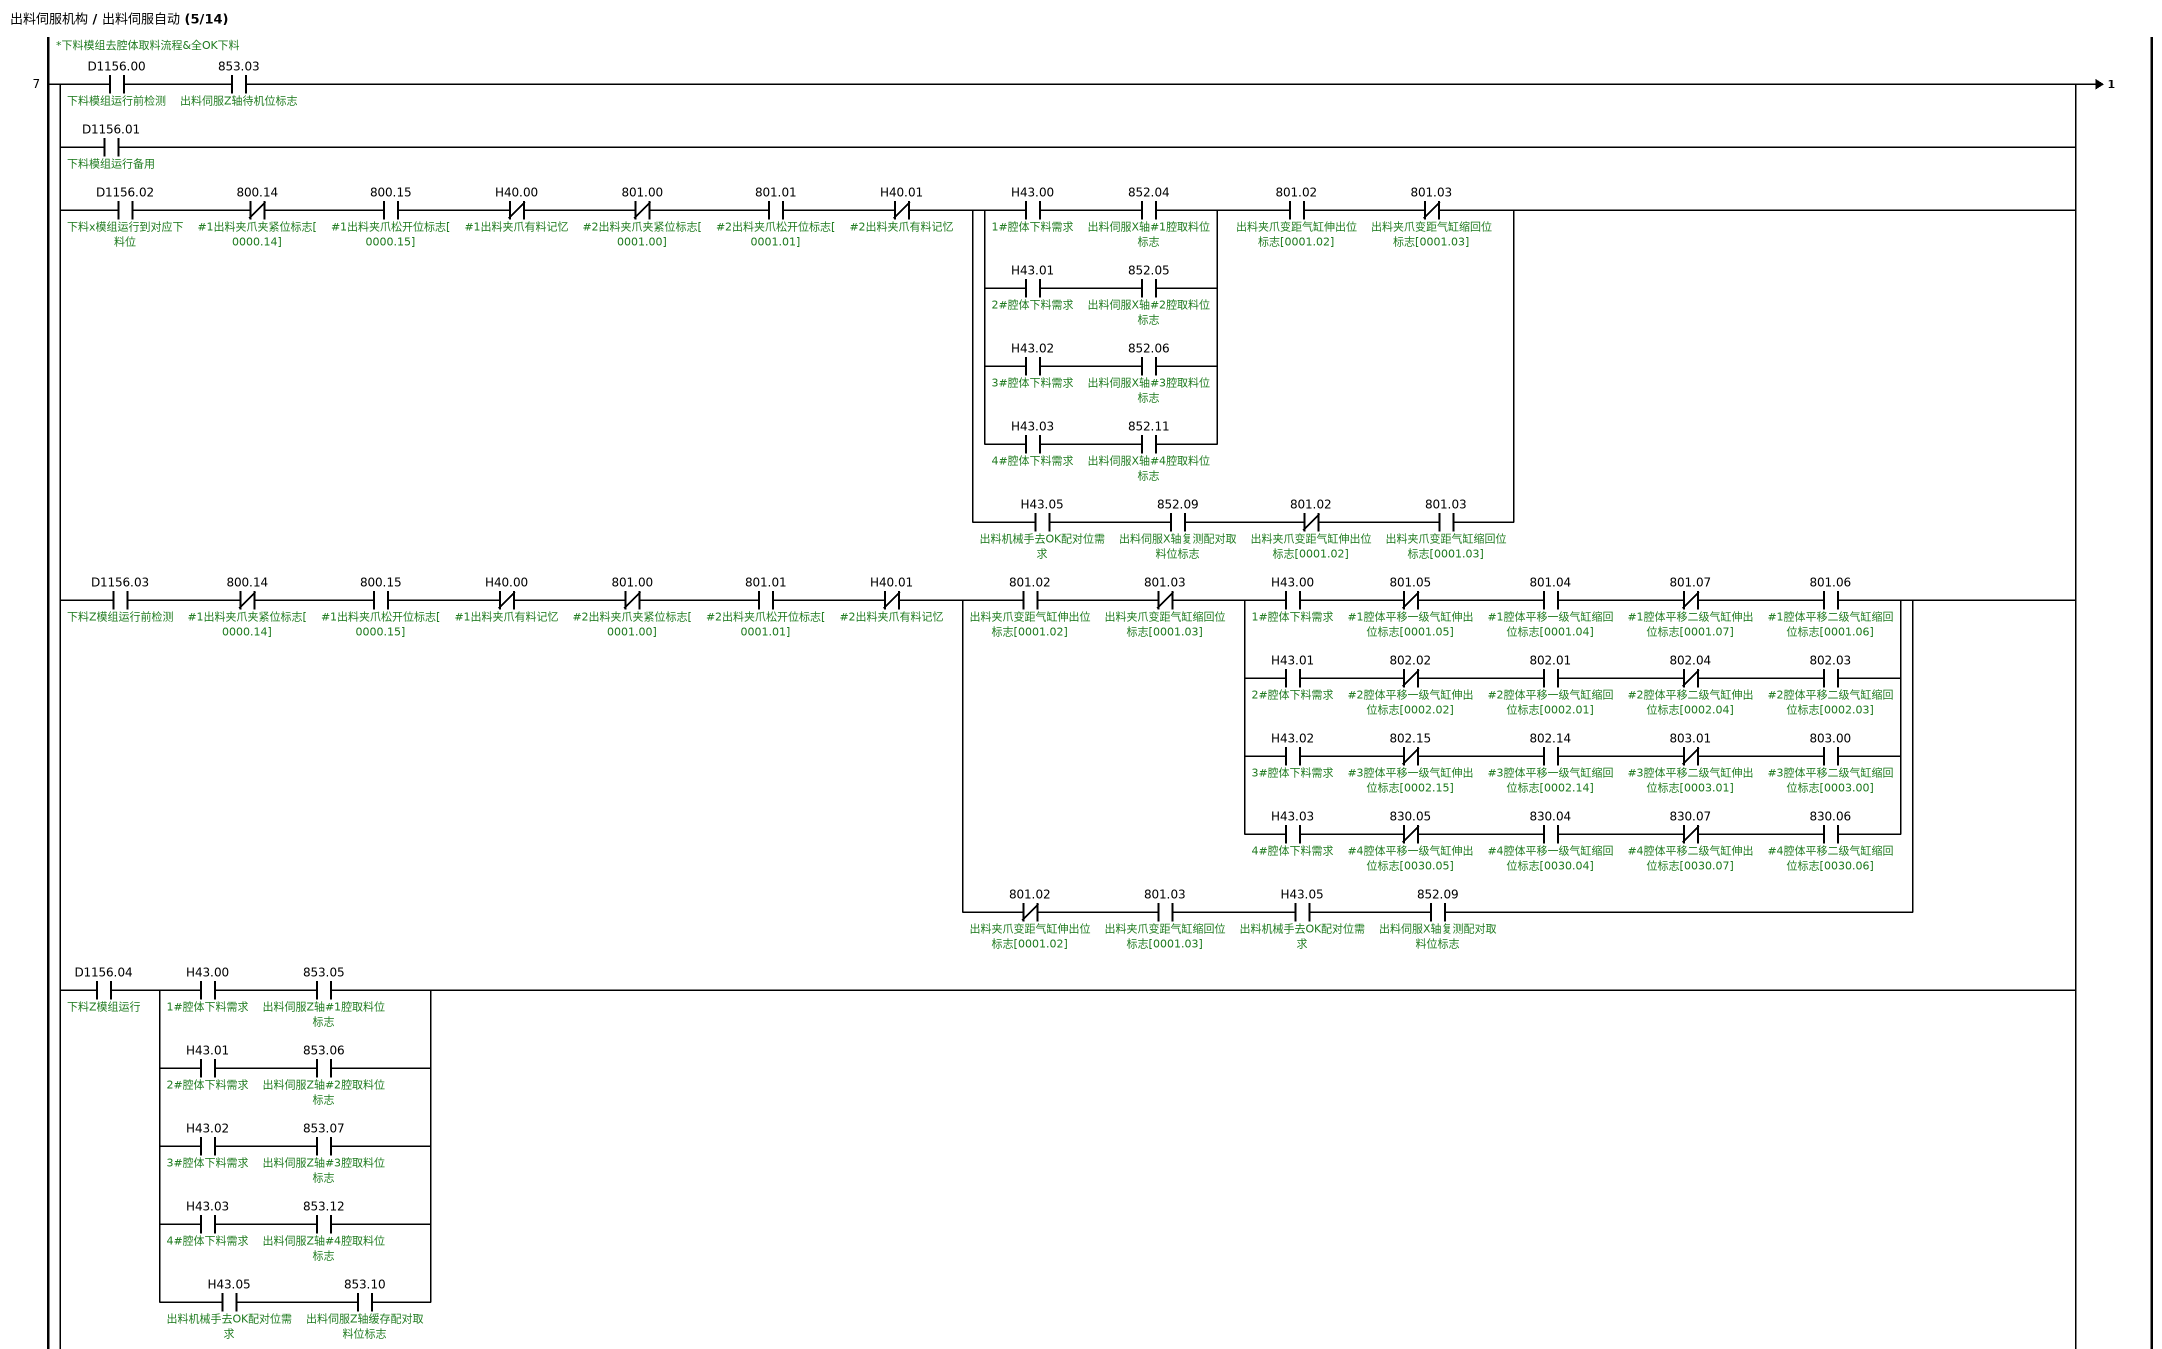

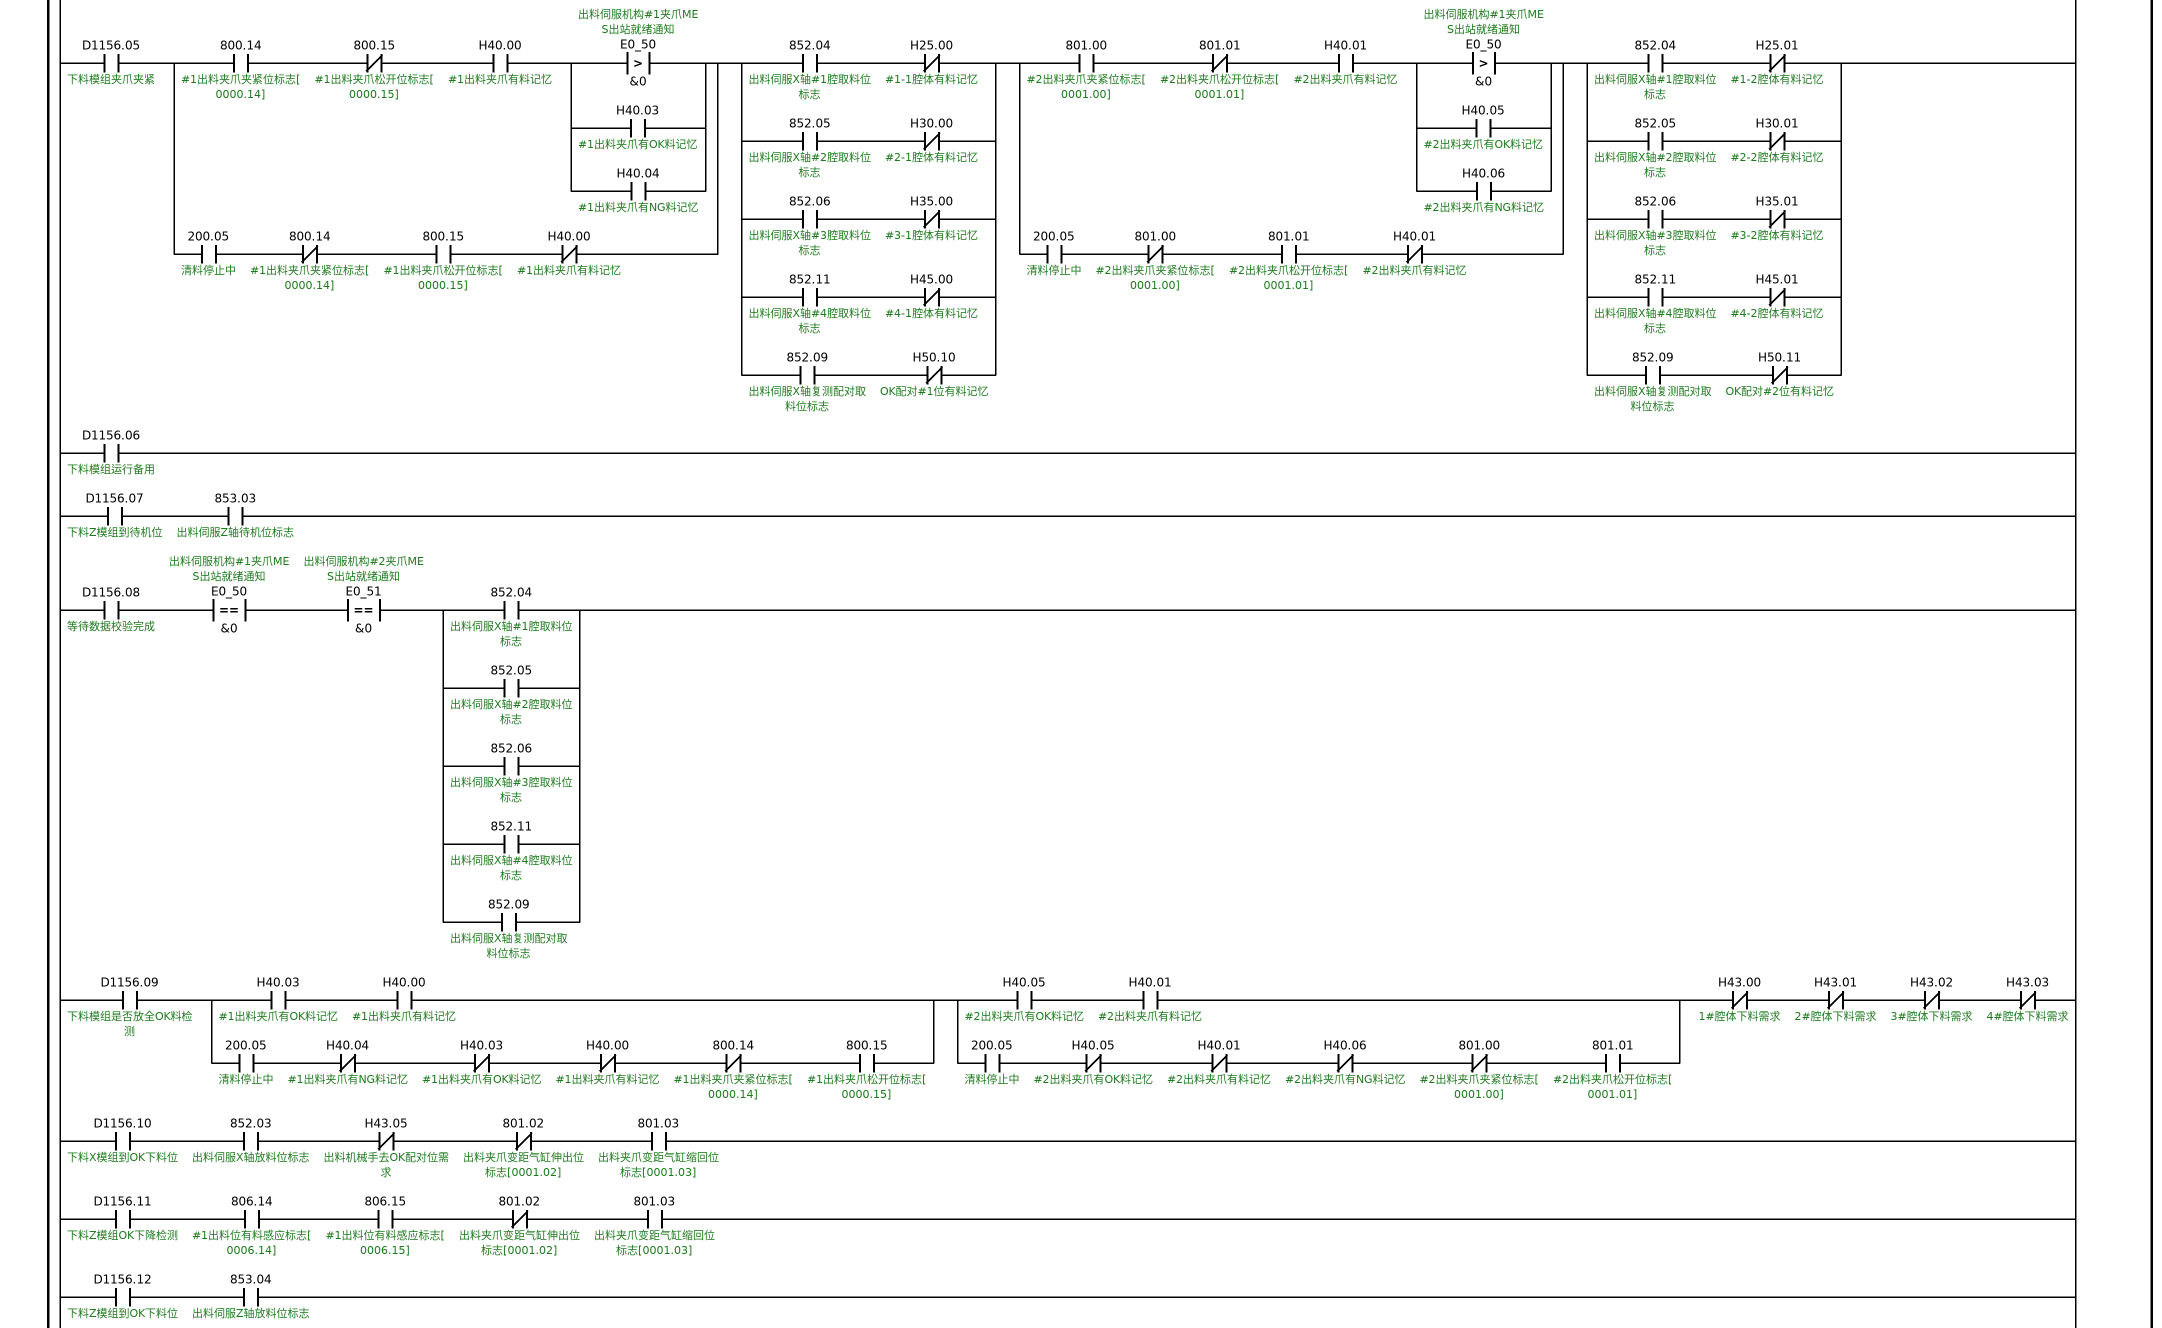

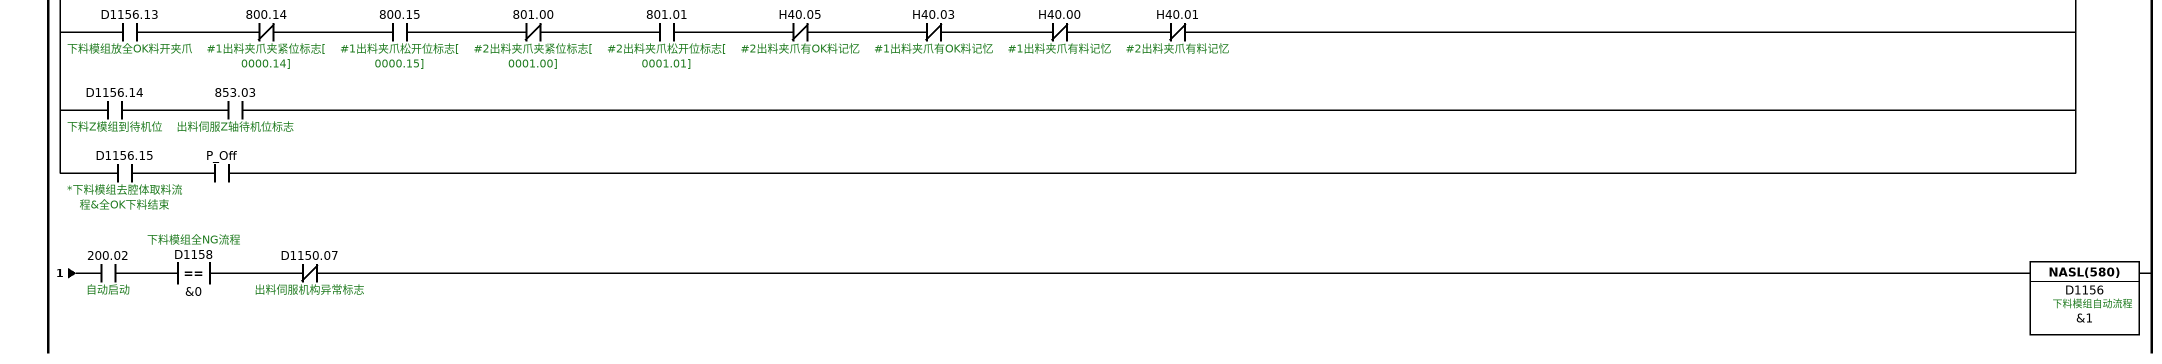
; rung 7: *下料模组去腔体取料流程&全OK下料
LD D1156.00  ; 下料模组运行前检测
AND 853.03  ; 出料伺服Z轴待机位标志
OR D1156.01  ; 下料模组运行备用
LD D1156.02  ; 下料x模组运行到对应下料位
ANDNOT 800.14  ; #1出料夹爪夹紧位标志[0000.14]
AND 800.15  ; #1出料夹爪松开位标志[0000.15]
ANDNOT H40.00  ; #1出料夹爪有料记忆
ANDNOT 801.00  ; #2出料夹爪夹紧位标志[0001.00]
AND 801.01  ; #2出料夹爪松开位标志[0001.01]
ANDNOT H40.01  ; #2出料夹爪有料记忆
LD H43.00  ; 1#腔体下料需求
AND 852.04  ; 出料伺服X轴#1腔取料位标志
LD H43.01  ; 2#腔体下料需求
AND 852.05  ; 出料伺服X轴#2腔取料位标志
ORLD
LD H43.02  ; 3#腔体下料需求
AND 852.06  ; 出料伺服X轴#3腔取料位标志
ORLD
LD H43.03  ; 4#腔体下料需求
AND 852.11  ; 出料伺服X轴#4腔取料位标志
ORLD
AND 801.02  ; 出料夹爪变距气缸伸出位标志[0001.02]
ANDNOT 801.03  ; 出料夹爪变距气缸缩回位标志[0001.03]
LD H43.05  ; 出料机械手去OK配对位需求
AND 852.09  ; 出料伺服X轴复测配对取料位标志
ANDNOT 801.02  ; 出料夹爪变距气缸伸出位标志[0001.02]
AND 801.03  ; 出料夹爪变距气缸缩回位标志[0001.03]
ORLD
ANDLD
ORLD
LD D1156.03  ; 下料Z模组运行前检测
ANDNOT 800.14  ; #1出料夹爪夹紧位标志[0000.14]
AND 800.15  ; #1出料夹爪松开位标志[0000.15]
ANDNOT H40.00  ; #1出料夹爪有料记忆
ANDNOT 801.00  ; #2出料夹爪夹紧位标志[0001.00]
AND 801.01  ; #2出料夹爪松开位标志[0001.01]
ANDNOT H40.01  ; #2出料夹爪有料记忆
LD 801.02  ; 出料夹爪变距气缸伸出位标志[0001.02]
ANDNOT 801.03  ; 出料夹爪变距气缸缩回位标志[0001.03]
LD H43.00  ; 1#腔体下料需求
ANDNOT 801.05  ; #1腔体平移一级气缸伸出位标志[0001.05]
AND 801.04  ; #1腔体平移一级气缸缩回位标志[0001.04]
ANDNOT 801.07  ; #1腔体平移二级气缸伸出位标志[0001.07]
AND 801.06  ; #1腔体平移二级气缸缩回位标志[0001.06]
LD H43.01  ; 2#腔体下料需求
ANDNOT 802.02  ; #2腔体平移一级气缸伸出位标志[0002.02]
AND 802.01  ; #2腔体平移一级气缸缩回位标志[0002.01]
ANDNOT 802.04  ; #2腔体平移二级气缸伸出位标志[0002.04]
AND 802.03  ; #2腔体平移二级气缸缩回位标志[0002.03]
ORLD
LD H43.02  ; 3#腔体下料需求
ANDNOT 802.15  ; #3腔体平移一级气缸伸出位标志[0002.15]
AND 802.14  ; #3腔体平移一级气缸缩回位标志[0002.14]
ANDNOT 803.01  ; #3腔体平移二级气缸伸出位标志[0003.01]
AND 803.00  ; #3腔体平移二级气缸缩回位标志[0003.00]
ORLD
LD H43.03  ; 4#腔体下料需求
ANDNOT 830.05  ; #4腔体平移一级气缸伸出位标志[0030.05]
AND 830.04  ; #4腔体平移一级气缸缩回位标志[0030.04]
ANDNOT 830.07  ; #4腔体平移二级气缸伸出位标志[0030.07]
AND 830.06  ; #4腔体平移二级气缸缩回位标志[0030.06]
ORLD
ANDLD
LDNOT 801.02  ; 出料夹爪变距气缸伸出位标志[0001.02]
AND 801.03  ; 出料夹爪变距气缸缩回位标志[0001.03]
AND H43.05  ; 出料机械手去OK配对位需求
AND 852.09  ; 出料伺服X轴复测配对取料位标志
ORLD
ANDLD
ORLD
LD D1156.04  ; 下料Z模组运行
LD H43.00  ; 1#腔体下料需求
AND 853.05  ; 出料伺服Z轴#1腔取料位标志
LD H43.01  ; 2#腔体下料需求
AND 853.06  ; 出料伺服Z轴#2腔取料位标志
ORLD
LD H43.02  ; 3#腔体下料需求
AND 853.07  ; 出料伺服Z轴#3腔取料位标志
ORLD
LD H43.03  ; 4#腔体下料需求
AND 853.12  ; 出料伺服Z轴#4腔取料位标志
ORLD
LD H43.05  ; 出料机械手去OK配对位需求
AND 853.10  ; 出料伺服Z轴缓存配对取料位标志
ORLD
ANDLD
ORLD
LD D1156.05  ; 下料模组夹爪夹紧
LD 800.14  ; #1出料夹爪夹紧位标志[0000.14]
ANDNOT 800.15  ; #1出料夹爪松开位标志[0000.15]
AND H40.00  ; #1出料夹爪有料记忆
LD>(320) E0_50 &0  ; 出料伺服机构#1夹爪MES出站就绪通知
OR H40.03  ; #1出料夹爪有OK料记忆
OR H40.04  ; #1出料夹爪有NG料记忆
ANDLD
LD 200.05  ; 清料停止中
ANDNOT 800.14  ; #1出料夹爪夹紧位标志[0000.14]
AND 800.15  ; #1出料夹爪松开位标志[0000.15]
ANDNOT H40.00  ; #1出料夹爪有料记忆
ORLD
ANDLD
LD 852.04  ; 出料伺服X轴#1腔取料位标志
ANDNOT H25.00  ; #1-1腔体有料记忆
LD 852.05  ; 出料伺服X轴#2腔取料位标志
ANDNOT H30.00  ; #2-1腔体有料记忆
ORLD
LD 852.06  ; 出料伺服X轴#3腔取料位标志
ANDNOT H35.00  ; #3-1腔体有料记忆
ORLD
LD 852.11  ; 出料伺服X轴#4腔取料位标志
ANDNOT H45.00  ; #4-1腔体有料记忆
ORLD
LD 852.09  ; 出料伺服X轴复测配对取料位标志
ANDNOT H50.10  ; OK配对#1位有料记忆
ORLD
ANDLD
LD 801.00  ; #2出料夹爪夹紧位标志[0001.00]
ANDNOT 801.01  ; #2出料夹爪松开位标志[0001.01]
AND H40.01  ; #2出料夹爪有料记忆
LD>(320) E0_50 &0  ; 出料伺服机构#1夹爪MES出站就绪通知
OR H40.05  ; #2出料夹爪有OK料记忆
OR H40.06  ; #2出料夹爪有NG料记忆
ANDLD
LD 200.05  ; 清料停止中
ANDNOT 801.00  ; #2出料夹爪夹紧位标志[0001.00]
AND 801.01  ; #2出料夹爪松开位标志[0001.01]
ANDNOT H40.01  ; #2出料夹爪有料记忆
ORLD
ANDLD
LD 852.04  ; 出料伺服X轴#1腔取料位标志
ANDNOT H25.01  ; #1-2腔体有料记忆
LD 852.05  ; 出料伺服X轴#2腔取料位标志
ANDNOT H30.01  ; #2-2腔体有料记忆
ORLD
LD 852.06  ; 出料伺服X轴#3腔取料位标志
ANDNOT H35.01  ; #3-2腔体有料记忆
ORLD
LD 852.11  ; 出料伺服X轴#4腔取料位标志
ANDNOT H45.01  ; #4-2腔体有料记忆
ORLD
LD 852.09  ; 出料伺服X轴复测配对取料位标志
ANDNOT H50.11  ; OK配对#2位有料记忆
ORLD
ANDLD
ORLD
OR D1156.06  ; 下料模组运行备用
LD D1156.07  ; 下料Z模组到待机位
AND 853.03  ; 出料伺服Z轴待机位标志
ORLD
LD D1156.08  ; 等待数据校验完成
AND=(300) E0_50 &0  ; 出料伺服机构#1夹爪MES出站就绪通知
AND=(300) E0_51 &0  ; 出料伺服机构#2夹爪MES出站就绪通知
LD 852.04  ; 出料伺服X轴#1腔取料位标志
OR 852.05  ; 出料伺服X轴#2腔取料位标志
OR 852.06  ; 出料伺服X轴#3腔取料位标志
OR 852.11  ; 出料伺服X轴#4腔取料位标志
OR 852.09  ; 出料伺服X轴复测配对取料位标志
ANDLD
ORLD
LD D1156.09  ; 下料模组是否放全OK料检测
LD H40.03  ; #1出料夹爪有OK料记忆
AND H40.00  ; #1出料夹爪有料记忆
LD 200.05  ; 清料停止中
ANDNOT H40.04  ; #1出料夹爪有NG料记忆
ANDNOT H40.03  ; #1出料夹爪有OK料记忆
ANDNOT H40.00  ; #1出料夹爪有料记忆
ANDNOT 800.14  ; #1出料夹爪夹紧位标志[0000.14]
AND 800.15  ; #1出料夹爪松开位标志[0000.15]
ORLD
ANDLD
LD H40.05  ; #2出料夹爪有OK料记忆
AND H40.01  ; #2出料夹爪有料记忆
LD 200.05  ; 清料停止中
ANDNOT H40.05  ; #2出料夹爪有OK料记忆
ANDNOT H40.01  ; #2出料夹爪有料记忆
ANDNOT H40.06  ; #2出料夹爪有NG料记忆
ANDNOT 801.00  ; #2出料夹爪夹紧位标志[0001.00]
AND 801.01  ; #2出料夹爪松开位标志[0001.01]
ORLD
ANDLD
ANDNOT H43.00  ; 1#腔体下料需求
ANDNOT H43.01  ; 2#腔体下料需求
ANDNOT H43.02  ; 3#腔体下料需求
ANDNOT H43.03  ; 4#腔体下料需求
ORLD
LD D1156.10  ; 下料X模组到OK下料位
AND 852.03  ; 出料伺服X轴放料位标志
ANDNOT H43.05  ; 出料机械手去OK配对位需求
ANDNOT 801.02  ; 出料夹爪变距气缸伸出位标志[0001.02]
AND 801.03  ; 出料夹爪变距气缸缩回位标志[0001.03]
ORLD
LD D1156.11  ; 下料Z模组OK下降检测
AND 806.14  ; #1出料位有料感应标志[0006.14]
AND 806.15  ; #1出料位有料感应标志[0006.15]
ANDNOT 801.02  ; 出料夹爪变距气缸伸出位标志[0001.02]
AND 801.03  ; 出料夹爪变距气缸缩回位标志[0001.03]
ORLD
LD D1156.12  ; 下料Z模组到OK下料位
AND 853.04  ; 出料伺服Z轴放料位标志
ORLD
LD D1156.13  ; 下料模组放全OK料开夹爪
ANDNOT 800.14  ; #1出料夹爪夹紧位标志[0000.14]
AND 800.15  ; #1出料夹爪松开位标志[0000.15]
ANDNOT 801.00  ; #2出料夹爪夹紧位标志[0001.00]
AND 801.01  ; #2出料夹爪松开位标志[0001.01]
ANDNOT H40.05  ; #2出料夹爪有OK料记忆
ANDNOT H40.03  ; #1出料夹爪有OK料记忆
ANDNOT H40.00  ; #1出料夹爪有料记忆
ANDNOT H40.01  ; #2出料夹爪有料记忆
ORLD
LD D1156.14  ; 下料Z模组到待机位
AND 853.03  ; 出料伺服Z轴待机位标志
ORLD
LD D1156.15  ; *下料模组去腔体取料流程&全OK下料结束
AND P_Off
ORLD
AND 200.02  ; 自动启动
AND=L(301) D1158 &0  ; 下料模组全NG流程
ANDNOT D1150.07  ; 出料伺服机构异常标志
NASL(580) D1156 &1  ; 下料模组自动流程

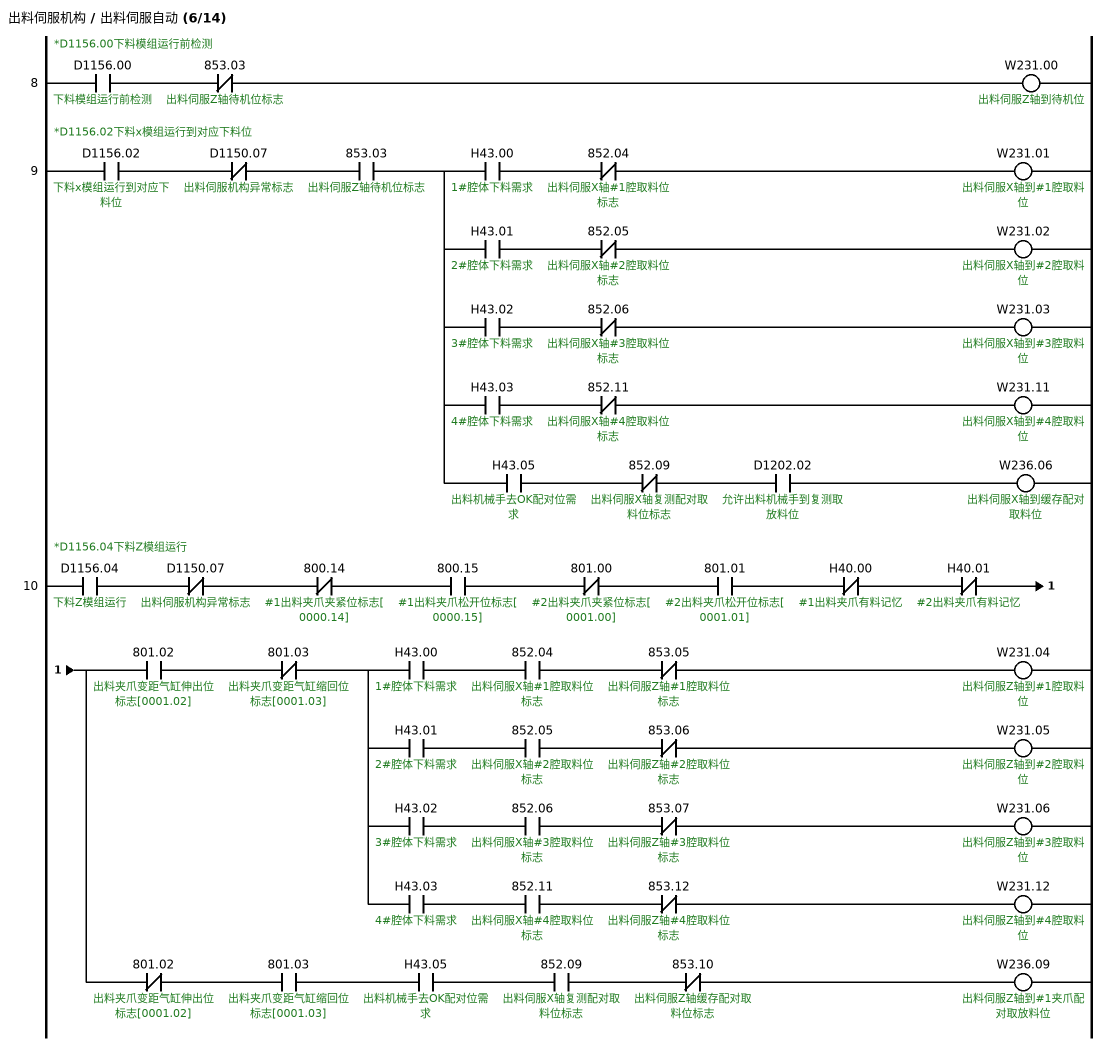
; rung 8: *D1156.00下料模组运行前检测
LD D1156.00  ; 下料模组运行前检测
ANDNOT 853.03  ; 出料伺服Z轴待机位标志
OUT W231.00  ; 出料伺服Z轴到待机位
; rung 9: *D1156.02下料x模组运行到对应下料位
LD D1156.02  ; 下料x模组运行到对应下料位
ANDNOT D1150.07  ; 出料伺服机构异常标志
AND 853.03  ; 出料伺服Z轴待机位标志
OUT TR0
AND H43.00  ; 1#腔体下料需求
ANDNOT 852.04  ; 出料伺服X轴#1腔取料位标志
OUT W231.01  ; 出料伺服X轴到#1腔取料位
LD TR0
AND H43.01  ; 2#腔体下料需求
ANDNOT 852.05  ; 出料伺服X轴#2腔取料位标志
OUT W231.02  ; 出料伺服X轴到#2腔取料位
LD TR0
AND H43.02  ; 3#腔体下料需求
ANDNOT 852.06  ; 出料伺服X轴#3腔取料位标志
OUT W231.03  ; 出料伺服X轴到#3腔取料位
LD TR0
AND H43.03  ; 4#腔体下料需求
ANDNOT 852.11  ; 出料伺服X轴#4腔取料位标志
OUT W231.11  ; 出料伺服X轴到#4腔取料位
LD TR0
AND H43.05  ; 出料机械手去OK配对位需求
ANDNOT 852.09  ; 出料伺服X轴复测配对取料位标志
AND D1202.02  ; 允许出料机械手到复测取放料位
OUT W236.06  ; 出料伺服X轴到缓存配对取料位
; rung 10: *D1156.04下料Z模组运行
LD D1156.04  ; 下料Z模组运行
ANDNOT D1150.07  ; 出料伺服机构异常标志
ANDNOT 800.14  ; #1出料夹爪夹紧位标志[0000.14]
AND 800.15  ; #1出料夹爪松开位标志[0000.15]
ANDNOT 801.00  ; #2出料夹爪夹紧位标志[0001.00]
AND 801.01  ; #2出料夹爪松开位标志[0001.01]
ANDNOT H40.00  ; #1出料夹爪有料记忆
ANDNOT H40.01  ; #2出料夹爪有料记忆
OUT TR0
AND 801.02  ; 出料夹爪变距气缸伸出位标志[0001.02]
ANDNOT 801.03  ; 出料夹爪变距气缸缩回位标志[0001.03]
OUT TR1
AND H43.00  ; 1#腔体下料需求
AND 852.04  ; 出料伺服X轴#1腔取料位标志
ANDNOT 853.05  ; 出料伺服Z轴#1腔取料位标志
OUT W231.04  ; 出料伺服Z轴到#1腔取料位
LD TR1
AND H43.01  ; 2#腔体下料需求
AND 852.05  ; 出料伺服X轴#2腔取料位标志
ANDNOT 853.06  ; 出料伺服Z轴#2腔取料位标志
OUT W231.05  ; 出料伺服Z轴到#2腔取料位
LD TR1
AND H43.02  ; 3#腔体下料需求
AND 852.06  ; 出料伺服X轴#3腔取料位标志
ANDNOT 853.07  ; 出料伺服Z轴#3腔取料位标志
OUT W231.06  ; 出料伺服Z轴到#3腔取料位
LD TR1
AND H43.03  ; 4#腔体下料需求
AND 852.11  ; 出料伺服X轴#4腔取料位标志
ANDNOT 853.12  ; 出料伺服Z轴#4腔取料位标志
OUT W231.12  ; 出料伺服Z轴到#4腔取料位
LD TR0
ANDNOT 801.02  ; 出料夹爪变距气缸伸出位标志[0001.02]
AND 801.03  ; 出料夹爪变距气缸缩回位标志[0001.03]
AND H43.05  ; 出料机械手去OK配对位需求
AND 852.09  ; 出料伺服X轴复测配对取料位标志
ANDNOT 853.10  ; 出料伺服Z轴缓存配对取料位标志
OUT W236.09  ; 出料伺服Z轴到#1夹爪配对取放料位

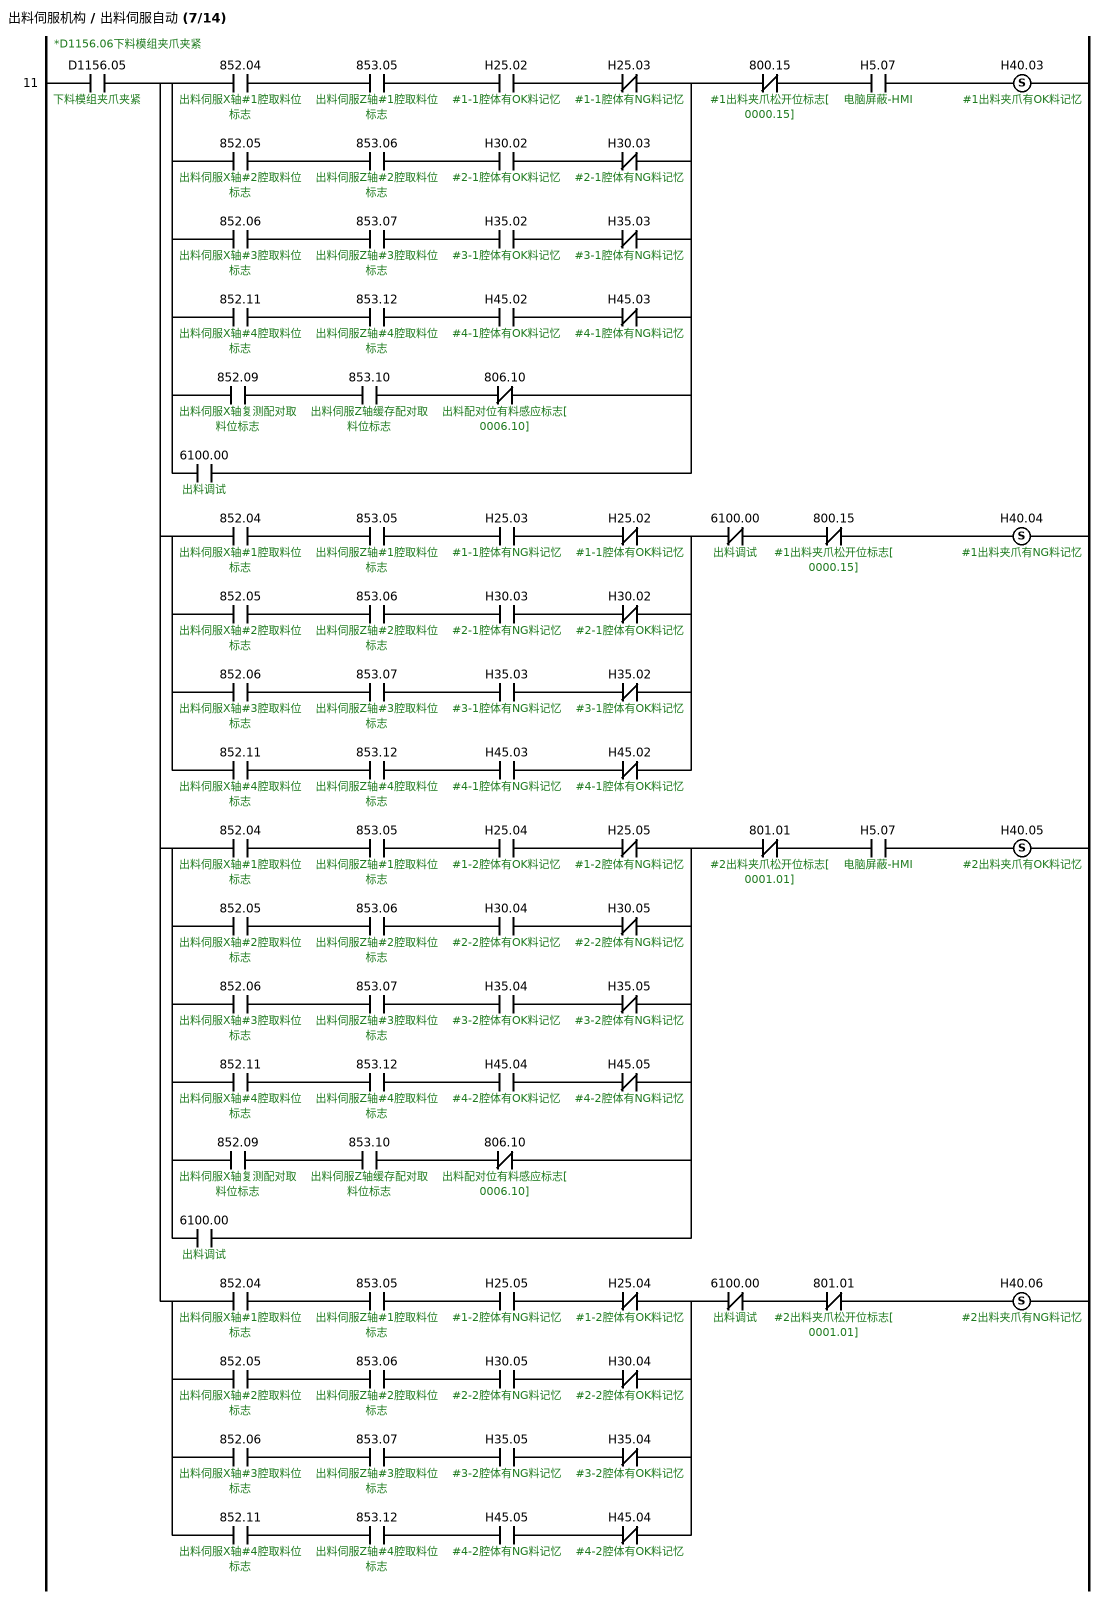
; rung 11: *D1156.06下料模组夹爪夹紧
LD D1156.05  ; 下料模组夹爪夹紧
OUT TR0
LD 852.04  ; 出料伺服X轴#1腔取料位标志
AND 853.05  ; 出料伺服Z轴#1腔取料位标志
AND H25.02  ; #1-1腔体有OK料记忆
ANDNOT H25.03  ; #1-1腔体有NG料记忆
LD 852.05  ; 出料伺服X轴#2腔取料位标志
AND 853.06  ; 出料伺服Z轴#2腔取料位标志
AND H30.02  ; #2-1腔体有OK料记忆
ANDNOT H30.03  ; #2-1腔体有NG料记忆
ORLD
LD 852.06  ; 出料伺服X轴#3腔取料位标志
AND 853.07  ; 出料伺服Z轴#3腔取料位标志
AND H35.02  ; #3-1腔体有OK料记忆
ANDNOT H35.03  ; #3-1腔体有NG料记忆
ORLD
LD 852.11  ; 出料伺服X轴#4腔取料位标志
AND 853.12  ; 出料伺服Z轴#4腔取料位标志
AND H45.02  ; #4-1腔体有OK料记忆
ANDNOT H45.03  ; #4-1腔体有NG料记忆
ORLD
LD 852.09  ; 出料伺服X轴复测配对取料位标志
AND 853.10  ; 出料伺服Z轴缓存配对取料位标志
ANDNOT 806.10  ; 出料配对位有料感应标志[0006.10]
ORLD
OR 6100.00  ; 出料调试
ANDLD
ANDNOT 800.15  ; #1出料夹爪松开位标志[0000.15]
AND H5.07  ; 电脑屏蔽-HMI
SET H40.03  ; #1出料夹爪有OK料记忆
LD TR0
LD 852.04  ; 出料伺服X轴#1腔取料位标志
AND 853.05  ; 出料伺服Z轴#1腔取料位标志
AND H25.03  ; #1-1腔体有NG料记忆
ANDNOT H25.02  ; #1-1腔体有OK料记忆
LD 852.05  ; 出料伺服X轴#2腔取料位标志
AND 853.06  ; 出料伺服Z轴#2腔取料位标志
AND H30.03  ; #2-1腔体有NG料记忆
ANDNOT H30.02  ; #2-1腔体有OK料记忆
ORLD
LD 852.06  ; 出料伺服X轴#3腔取料位标志
AND 853.07  ; 出料伺服Z轴#3腔取料位标志
AND H35.03  ; #3-1腔体有NG料记忆
ANDNOT H35.02  ; #3-1腔体有OK料记忆
ORLD
LD 852.11  ; 出料伺服X轴#4腔取料位标志
AND 853.12  ; 出料伺服Z轴#4腔取料位标志
AND H45.03  ; #4-1腔体有NG料记忆
ANDNOT H45.02  ; #4-1腔体有OK料记忆
ORLD
ANDLD
ANDNOT 6100.00  ; 出料调试
ANDNOT 800.15  ; #1出料夹爪松开位标志[0000.15]
SET H40.04  ; #1出料夹爪有NG料记忆
LD TR0
LD 852.04  ; 出料伺服X轴#1腔取料位标志
AND 853.05  ; 出料伺服Z轴#1腔取料位标志
AND H25.04  ; #1-2腔体有OK料记忆
ANDNOT H25.05  ; #1-2腔体有NG料记忆
LD 852.05  ; 出料伺服X轴#2腔取料位标志
AND 853.06  ; 出料伺服Z轴#2腔取料位标志
AND H30.04  ; #2-2腔体有OK料记忆
ANDNOT H30.05  ; #2-2腔体有NG料记忆
ORLD
LD 852.06  ; 出料伺服X轴#3腔取料位标志
AND 853.07  ; 出料伺服Z轴#3腔取料位标志
AND H35.04  ; #3-2腔体有OK料记忆
ANDNOT H35.05  ; #3-2腔体有NG料记忆
ORLD
LD 852.11  ; 出料伺服X轴#4腔取料位标志
AND 853.12  ; 出料伺服Z轴#4腔取料位标志
AND H45.04  ; #4-2腔体有OK料记忆
ANDNOT H45.05  ; #4-2腔体有NG料记忆
ORLD
LD 852.09  ; 出料伺服X轴复测配对取料位标志
AND 853.10  ; 出料伺服Z轴缓存配对取料位标志
ANDNOT 806.10  ; 出料配对位有料感应标志[0006.10]
ORLD
OR 6100.00  ; 出料调试
ANDLD
ANDNOT 801.01  ; #2出料夹爪松开位标志[0001.01]
AND H5.07  ; 电脑屏蔽-HMI
SET H40.05  ; #2出料夹爪有OK料记忆
LD TR0
LD 852.04  ; 出料伺服X轴#1腔取料位标志
AND 853.05  ; 出料伺服Z轴#1腔取料位标志
AND H25.05  ; #1-2腔体有NG料记忆
ANDNOT H25.04  ; #1-2腔体有OK料记忆
LD 852.05  ; 出料伺服X轴#2腔取料位标志
AND 853.06  ; 出料伺服Z轴#2腔取料位标志
AND H30.05  ; #2-2腔体有NG料记忆
ANDNOT H30.04  ; #2-2腔体有OK料记忆
ORLD
LD 852.06  ; 出料伺服X轴#3腔取料位标志
AND 853.07  ; 出料伺服Z轴#3腔取料位标志
AND H35.05  ; #3-2腔体有NG料记忆
ANDNOT H35.04  ; #3-2腔体有OK料记忆
ORLD
LD 852.11  ; 出料伺服X轴#4腔取料位标志
AND 853.12  ; 出料伺服Z轴#4腔取料位标志
AND H45.05  ; #4-2腔体有NG料记忆
ANDNOT H45.04  ; #4-2腔体有OK料记忆
ORLD
ANDLD
ANDNOT 6100.00  ; 出料调试
ANDNOT 801.01  ; #2出料夹爪松开位标志[0001.01]
SET H40.06  ; #2出料夹爪有NG料记忆

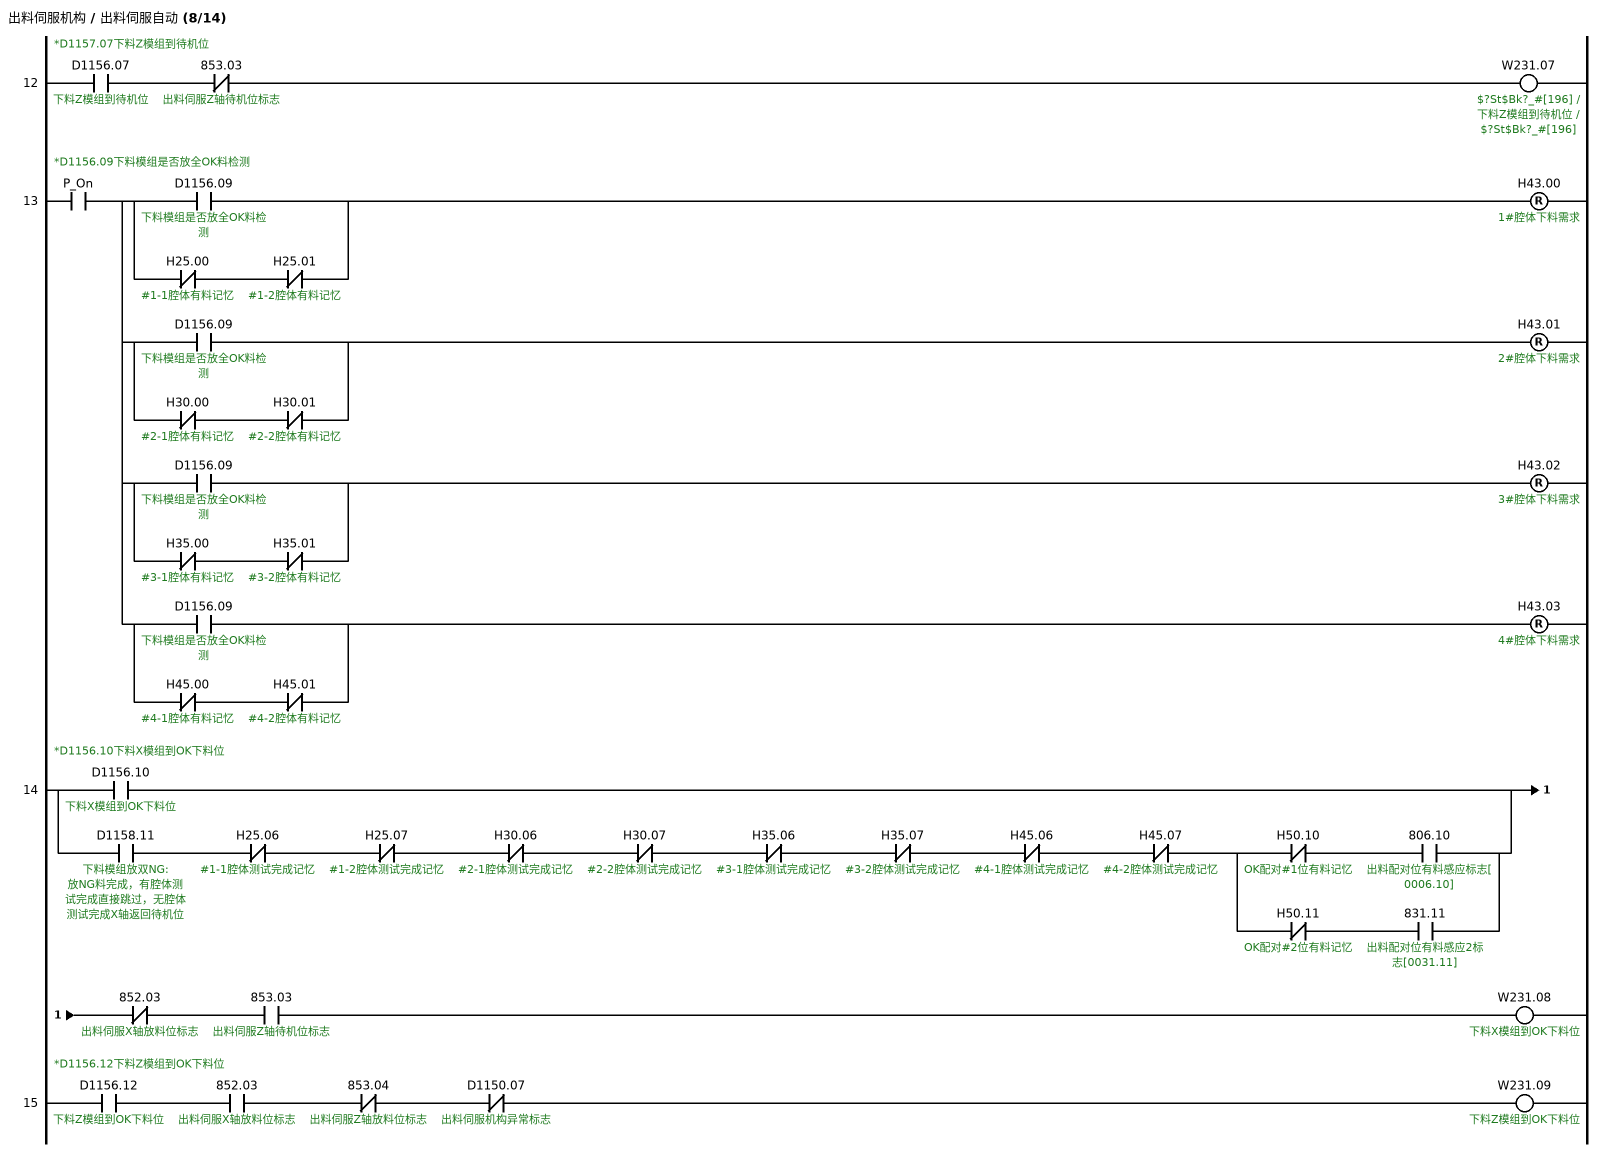
; rung 12: *D1157.07下料Z模组到待机位
LD D1156.07  ; 下料Z模组到待机位
ANDNOT 853.03  ; 出料伺服Z轴待机位标志
OUT W231.07  ; $?St$Bk?_#[196] / 下料Z模组到待机位 / $?St$Bk?_#[196]
; rung 13: *D1156.09下料模组是否放全OK料检测
LD P_On
OUT TR0
LD D1156.09  ; 下料模组是否放全OK料检测
LDNOT H25.00  ; #1-1腔体有料记忆
ANDNOT H25.01  ; #1-2腔体有料记忆
ORLD
ANDLD
RSET H43.00  ; 1#腔体下料需求
LD TR0
LD D1156.09  ; 下料模组是否放全OK料检测
LDNOT H30.00  ; #2-1腔体有料记忆
ANDNOT H30.01  ; #2-2腔体有料记忆
ORLD
ANDLD
RSET H43.01  ; 2#腔体下料需求
LD TR0
LD D1156.09  ; 下料模组是否放全OK料检测
LDNOT H35.00  ; #3-1腔体有料记忆
ANDNOT H35.01  ; #3-2腔体有料记忆
ORLD
ANDLD
RSET H43.02  ; 3#腔体下料需求
LD TR0
LD D1156.09  ; 下料模组是否放全OK料检测
LDNOT H45.00  ; #4-1腔体有料记忆
ANDNOT H45.01  ; #4-2腔体有料记忆
ORLD
ANDLD
RSET H43.03  ; 4#腔体下料需求
; rung 14: *D1156.10下料X模组到OK下料位
LD D1156.10  ; 下料X模组到OK下料位
LD D1158.11  ; 下料模组放双NG:放NG料完成，有腔体测试完成直接跳过，无腔体测试完成X轴返回待机位
ANDNOT H25.06  ; #1-1腔体测试完成记忆
ANDNOT H25.07  ; #1-2腔体测试完成记忆
ANDNOT H30.06  ; #2-1腔体测试完成记忆
ANDNOT H30.07  ; #2-2腔体测试完成记忆
ANDNOT H35.06  ; #3-1腔体测试完成记忆
ANDNOT H35.07  ; #3-2腔体测试完成记忆
ANDNOT H45.06  ; #4-1腔体测试完成记忆
ANDNOT H45.07  ; #4-2腔体测试完成记忆
LDNOT H50.10  ; OK配对#1位有料记忆
AND 806.10  ; 出料配对位有料感应标志[0006.10]
LDNOT H50.11  ; OK配对#2位有料记忆
AND 831.11  ; 出料配对位有料感应2标志[0031.11]
ORLD
ANDLD
ORLD
ANDNOT 852.03  ; 出料伺服X轴放料位标志
AND 853.03  ; 出料伺服Z轴待机位标志
OUT W231.08  ; 下料X模组到OK下料位
; rung 15: *D1156.12下料Z模组到OK下料位
LD D1156.12  ; 下料Z模组到OK下料位
AND 852.03  ; 出料伺服X轴放料位标志
ANDNOT 853.04  ; 出料伺服Z轴放料位标志
ANDNOT D1150.07  ; 出料伺服机构异常标志
OUT W231.09  ; 下料Z模组到OK下料位

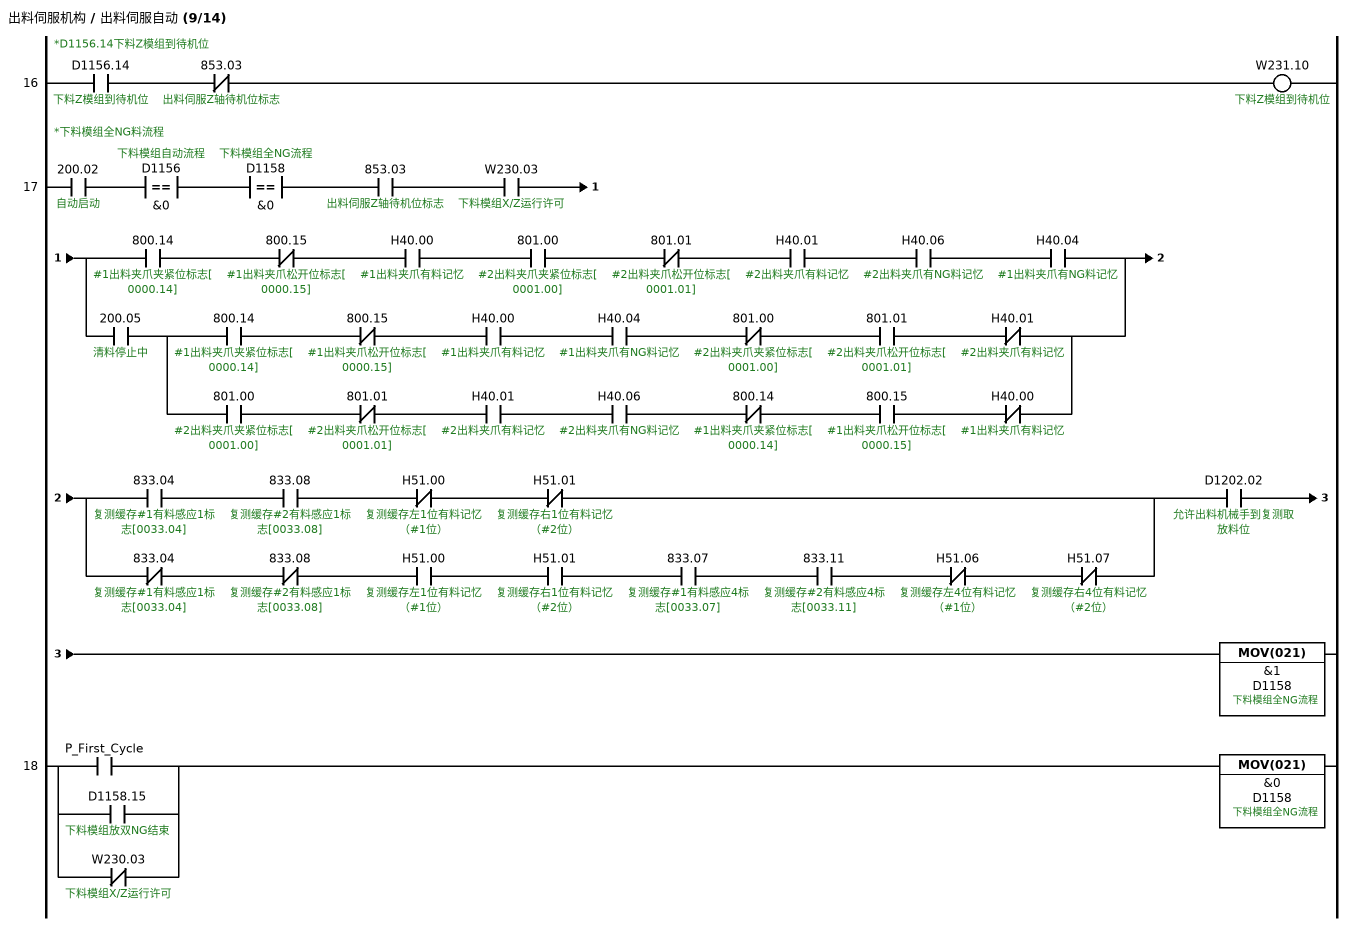
; rung 16: *D1156.14下料Z模组到待机位
LD D1156.14  ; 下料Z模组到待机位
ANDNOT 853.03  ; 出料伺服Z轴待机位标志
OUT W231.10  ; 下料Z模组到待机位
; rung 17: *下料模组全NG料流程
LD 200.02  ; 自动启动
AND=L(301) D1156 &0  ; 下料模组自动流程
AND=L(301) D1158 &0  ; 下料模组全NG流程
AND 853.03  ; 出料伺服Z轴待机位标志
AND W230.03  ; 下料模组X/Z运行许可
LD 800.14  ; #1出料夹爪夹紧位标志[0000.14]
ANDNOT 800.15  ; #1出料夹爪松开位标志[0000.15]
AND H40.00  ; #1出料夹爪有料记忆
AND 801.00  ; #2出料夹爪夹紧位标志[0001.00]
ANDNOT 801.01  ; #2出料夹爪松开位标志[0001.01]
AND H40.01  ; #2出料夹爪有料记忆
AND H40.06  ; #2出料夹爪有NG料记忆
AND H40.04  ; #1出料夹爪有NG料记忆
LD 200.05  ; 清料停止中
LD 800.14  ; #1出料夹爪夹紧位标志[0000.14]
ANDNOT 800.15  ; #1出料夹爪松开位标志[0000.15]
AND H40.00  ; #1出料夹爪有料记忆
AND H40.04  ; #1出料夹爪有NG料记忆
ANDNOT 801.00  ; #2出料夹爪夹紧位标志[0001.00]
AND 801.01  ; #2出料夹爪松开位标志[0001.01]
ANDNOT H40.01  ; #2出料夹爪有料记忆
LD 801.00  ; #2出料夹爪夹紧位标志[0001.00]
ANDNOT 801.01  ; #2出料夹爪松开位标志[0001.01]
AND H40.01  ; #2出料夹爪有料记忆
AND H40.06  ; #2出料夹爪有NG料记忆
ANDNOT 800.14  ; #1出料夹爪夹紧位标志[0000.14]
AND 800.15  ; #1出料夹爪松开位标志[0000.15]
ANDNOT H40.00  ; #1出料夹爪有料记忆
ORLD
ANDLD
ORLD
ANDLD
LD 833.04  ; 复测缓存#1有料感应1标志[0033.04]
AND 833.08  ; 复测缓存#2有料感应1标志[0033.08]
ANDNOT H51.00  ; 复测缓存左1位有料记忆（#1位）
ANDNOT H51.01  ; 复测缓存右1位有料记忆（#2位）
LDNOT 833.04  ; 复测缓存#1有料感应1标志[0033.04]
ANDNOT 833.08  ; 复测缓存#2有料感应1标志[0033.08]
AND H51.00  ; 复测缓存左1位有料记忆（#1位）
AND H51.01  ; 复测缓存右1位有料记忆（#2位）
AND 833.07  ; 复测缓存#1有料感应4标志[0033.07]
AND 833.11  ; 复测缓存#2有料感应4标志[0033.11]
ANDNOT H51.06  ; 复测缓存左4位有料记忆（#1位）
ANDNOT H51.07  ; 复测缓存右4位有料记忆（#2位）
ORLD
ANDLD
AND D1202.02  ; 允许出料机械手到复测取放料位
MOV(021) &1 D1158  ; 下料模组全NG流程
; rung 18
LD P_First_Cycle
OR D1158.15  ; 下料模组放双NG结束
ORNOT W230.03  ; 下料模组X/Z运行许可
MOV(021) &0 D1158  ; 下料模组全NG流程

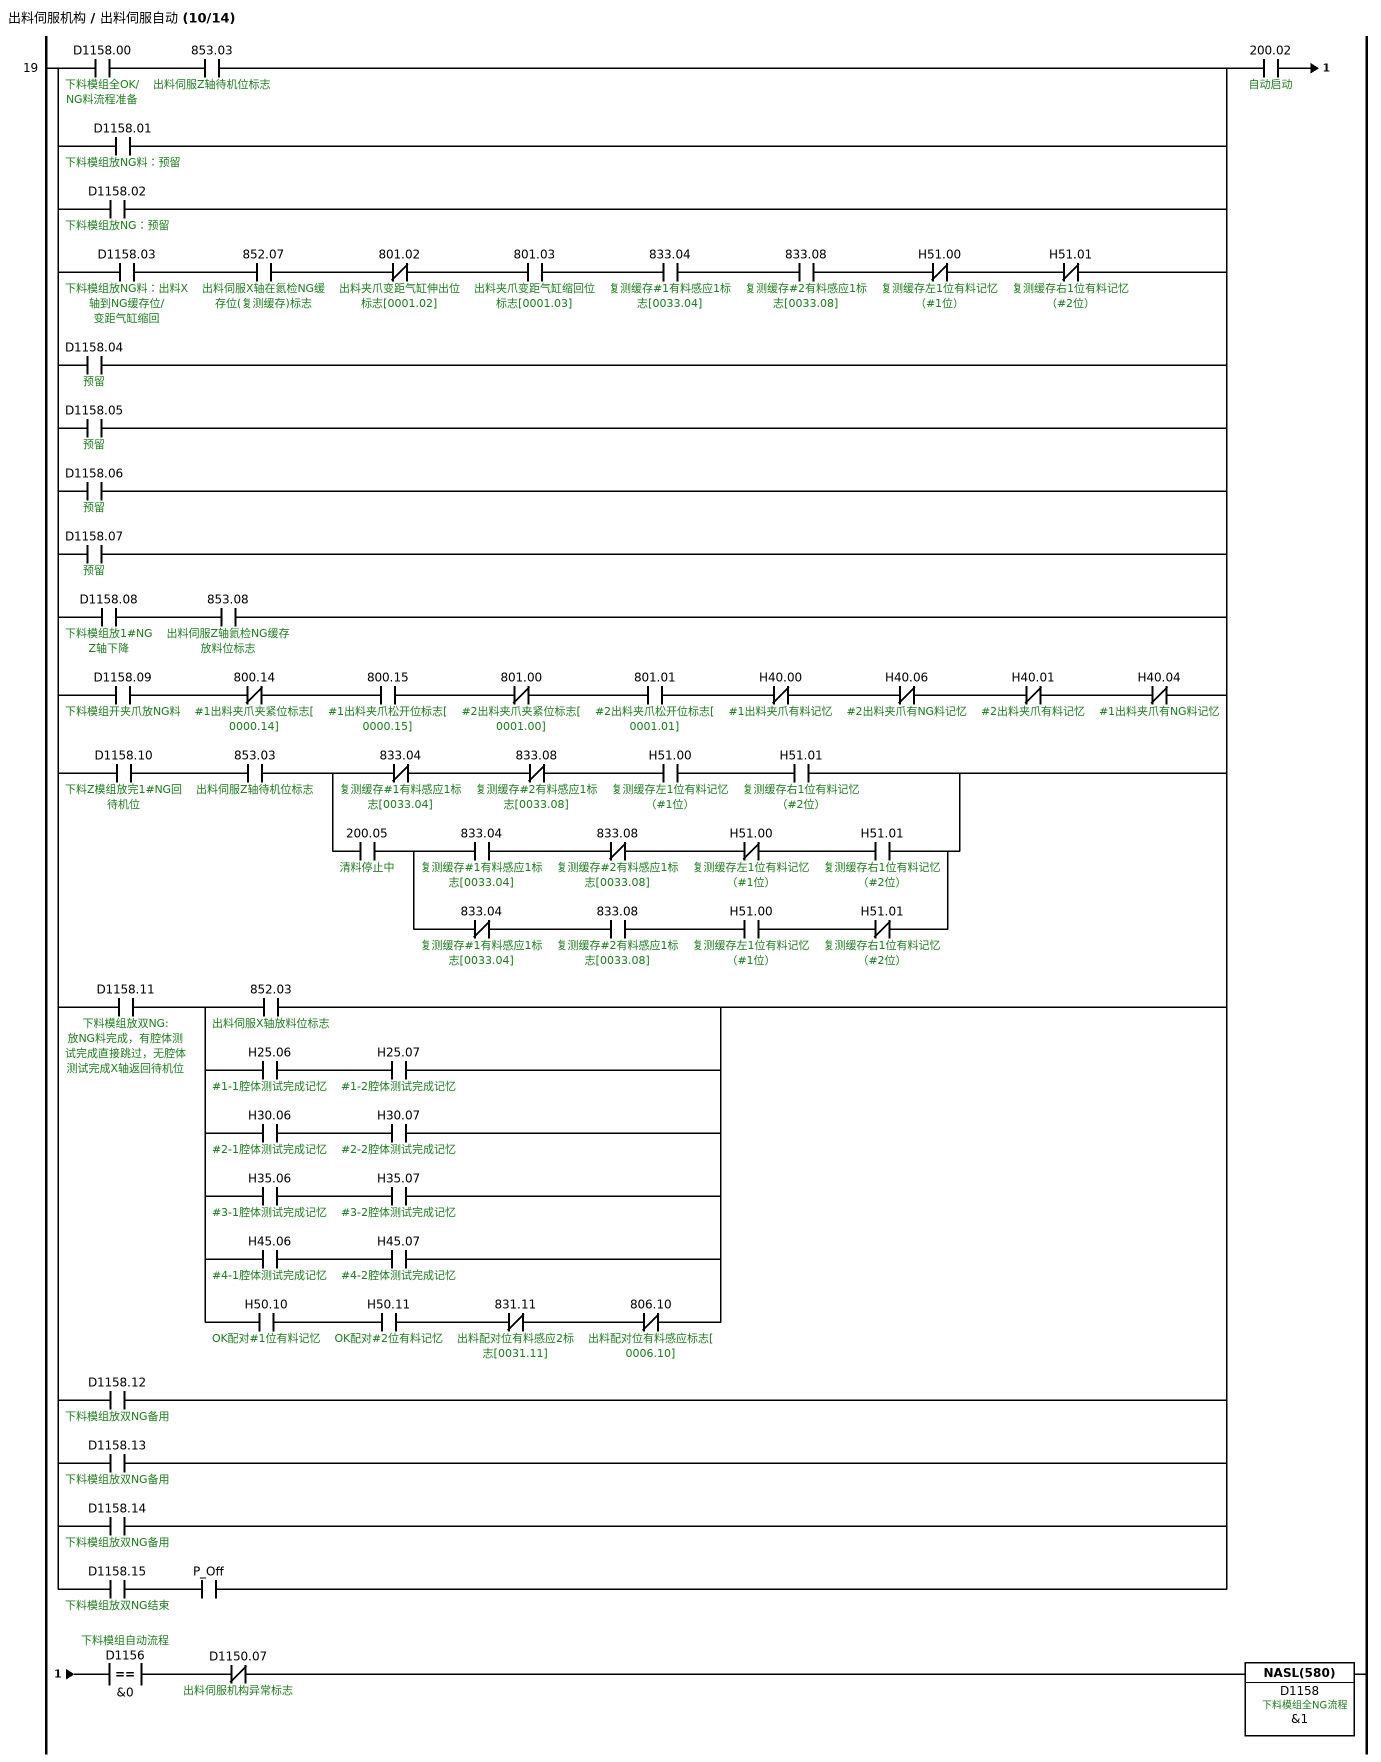
; rung 19
LD D1158.00  ; 下料模组全OK/NG料流程准备
AND 853.03  ; 出料伺服Z轴待机位标志
OR D1158.01  ; 下料模组放NG料：预留
OR D1158.02  ; 下料模组放NG：预留
LD D1158.03  ; 下料模组放NG料：出料X轴到NG缓存位/变距气缸缩回
AND 852.07  ; 出料伺服X轴在氦检NG缓存位(复测缓存)标志
ANDNOT 801.02  ; 出料夹爪变距气缸伸出位标志[0001.02]
AND 801.03  ; 出料夹爪变距气缸缩回位标志[0001.03]
AND 833.04  ; 复测缓存#1有料感应1标志[0033.04]
AND 833.08  ; 复测缓存#2有料感应1标志[0033.08]
ANDNOT H51.00  ; 复测缓存左1位有料记忆（#1位）
ANDNOT H51.01  ; 复测缓存右1位有料记忆（#2位）
ORLD
OR D1158.04  ; 预留
OR D1158.05  ; 预留
OR D1158.06  ; 预留
OR D1158.07  ; 预留
LD D1158.08  ; 下料模组放1#NG Z轴下降
AND 853.08  ; 出料伺服Z轴氦检NG缓存放料位标志
ORLD
LD D1158.09  ; 下料模组开夹爪放NG料
ANDNOT 800.14  ; #1出料夹爪夹紧位标志[0000.14]
AND 800.15  ; #1出料夹爪松开位标志[0000.15]
ANDNOT 801.00  ; #2出料夹爪夹紧位标志[0001.00]
AND 801.01  ; #2出料夹爪松开位标志[0001.01]
ANDNOT H40.00  ; #1出料夹爪有料记忆
ANDNOT H40.06  ; #2出料夹爪有NG料记忆
ANDNOT H40.01  ; #2出料夹爪有料记忆
ANDNOT H40.04  ; #1出料夹爪有NG料记忆
ORLD
LD D1158.10  ; 下料Z模组放完1#NG回待机位
AND 853.03  ; 出料伺服Z轴待机位标志
LDNOT 833.04  ; 复测缓存#1有料感应1标志[0033.04]
ANDNOT 833.08  ; 复测缓存#2有料感应1标志[0033.08]
AND H51.00  ; 复测缓存左1位有料记忆（#1位）
AND H51.01  ; 复测缓存右1位有料记忆（#2位）
LD 200.05  ; 清料停止中
LD 833.04  ; 复测缓存#1有料感应1标志[0033.04]
ANDNOT 833.08  ; 复测缓存#2有料感应1标志[0033.08]
ANDNOT H51.00  ; 复测缓存左1位有料记忆（#1位）
AND H51.01  ; 复测缓存右1位有料记忆（#2位）
LDNOT 833.04  ; 复测缓存#1有料感应1标志[0033.04]
AND 833.08  ; 复测缓存#2有料感应1标志[0033.08]
AND H51.00  ; 复测缓存左1位有料记忆（#1位）
ANDNOT H51.01  ; 复测缓存右1位有料记忆（#2位）
ORLD
ANDLD
ORLD
ANDLD
ORLD
LD D1158.11  ; 下料模组放双NG:放NG料完成，有腔体测试完成直接跳过，无腔体测试完成X轴返回待机位
LD 852.03  ; 出料伺服X轴放料位标志
LD H25.06  ; #1-1腔体测试完成记忆
AND H25.07  ; #1-2腔体测试完成记忆
ORLD
LD H30.06  ; #2-1腔体测试完成记忆
AND H30.07  ; #2-2腔体测试完成记忆
ORLD
LD H35.06  ; #3-1腔体测试完成记忆
AND H35.07  ; #3-2腔体测试完成记忆
ORLD
LD H45.06  ; #4-1腔体测试完成记忆
AND H45.07  ; #4-2腔体测试完成记忆
ORLD
LD H50.10  ; OK配对#1位有料记忆
AND H50.11  ; OK配对#2位有料记忆
ANDNOT 831.11  ; 出料配对位有料感应2标志[0031.11]
ANDNOT 806.10  ; 出料配对位有料感应标志[0006.10]
ORLD
ANDLD
ORLD
OR D1158.12  ; 下料模组放双NG备用
OR D1158.13  ; 下料模组放双NG备用
OR D1158.14  ; 下料模组放双NG备用
LD D1158.15  ; 下料模组放双NG结束
AND P_Off
ORLD
AND 200.02  ; 自动启动
AND=L(301) D1156 &0  ; 下料模组自动流程
ANDNOT D1150.07  ; 出料伺服机构异常标志
NASL(580) D1158 &1  ; 下料模组全NG流程

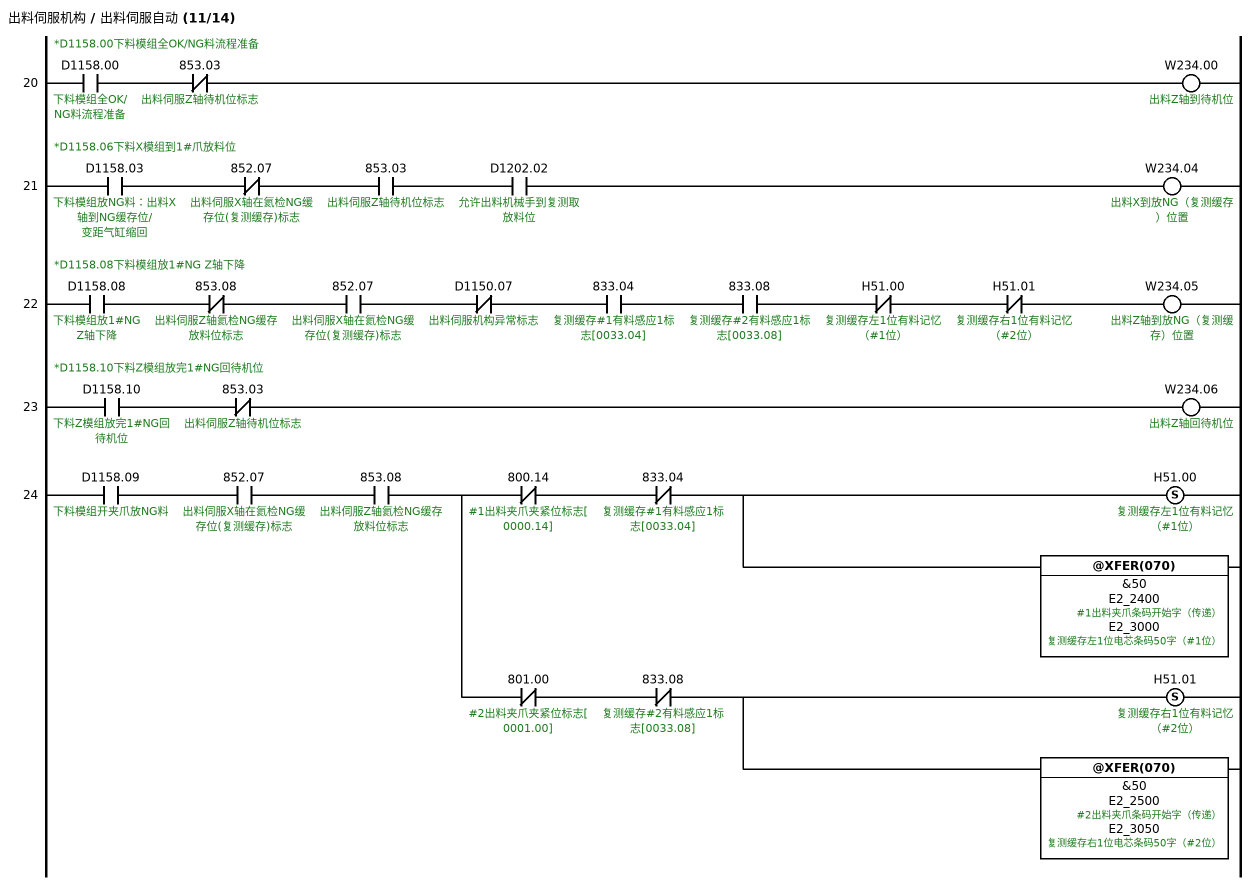
; rung 20: *D1158.00下料模组全OK/NG料流程准备
LD D1158.00  ; 下料模组全OK/NG料流程准备
ANDNOT 853.03  ; 出料伺服Z轴待机位标志
OUT W234.00  ; 出料Z轴到待机位
; rung 21: *D1158.06下料X模组到1#爪放料位
LD D1158.03  ; 下料模组放NG料：出料X轴到NG缓存位/变距气缸缩回
ANDNOT 852.07  ; 出料伺服X轴在氦检NG缓存位(复测缓存)标志
AND 853.03  ; 出料伺服Z轴待机位标志
AND D1202.02  ; 允许出料机械手到复测取放料位
OUT W234.04  ; 出料X到放NG（复测缓存）位置
; rung 22: *D1158.08下料模组放1#NG Z轴下降
LD D1158.08  ; 下料模组放1#NG Z轴下降
ANDNOT 853.08  ; 出料伺服Z轴氦检NG缓存放料位标志
AND 852.07  ; 出料伺服X轴在氦检NG缓存位(复测缓存)标志
ANDNOT D1150.07  ; 出料伺服机构异常标志
AND 833.04  ; 复测缓存#1有料感应1标志[0033.04]
AND 833.08  ; 复测缓存#2有料感应1标志[0033.08]
ANDNOT H51.00  ; 复测缓存左1位有料记忆（#1位）
ANDNOT H51.01  ; 复测缓存右1位有料记忆（#2位）
OUT W234.05  ; 出料Z轴到放NG（复测缓存）位置
; rung 23: *D1158.10下料Z模组放完1#NG回待机位
LD D1158.10  ; 下料Z模组放完1#NG回待机位
ANDNOT 853.03  ; 出料伺服Z轴待机位标志
OUT W234.06  ; 出料Z轴回待机位
; rung 24
LD D1158.09  ; 下料模组开夹爪放NG料
AND 852.07  ; 出料伺服X轴在氦检NG缓存位(复测缓存)标志
AND 853.08  ; 出料伺服Z轴氦检NG缓存放料位标志
OUT TR0
ANDNOT 800.14  ; #1出料夹爪夹紧位标志[0000.14]
ANDNOT 833.04  ; 复测缓存#1有料感应1标志[0033.04]
SET H51.00  ; 复测缓存左1位有料记忆（#1位）
@XFER(070) &50 E2_2400 E2_3000  ; #1出料夹爪条码开始字（传递）, 复测缓存左1位电芯条码50字（#1位）
LD TR0
ANDNOT 801.00  ; #2出料夹爪夹紧位标志[0001.00]
ANDNOT 833.08  ; 复测缓存#2有料感应1标志[0033.08]
SET H51.01  ; 复测缓存右1位有料记忆（#2位）
@XFER(070) &50 E2_2500 E2_3050  ; #2出料夹爪条码开始字（传递）, 复测缓存右1位电芯条码50字（#2位）

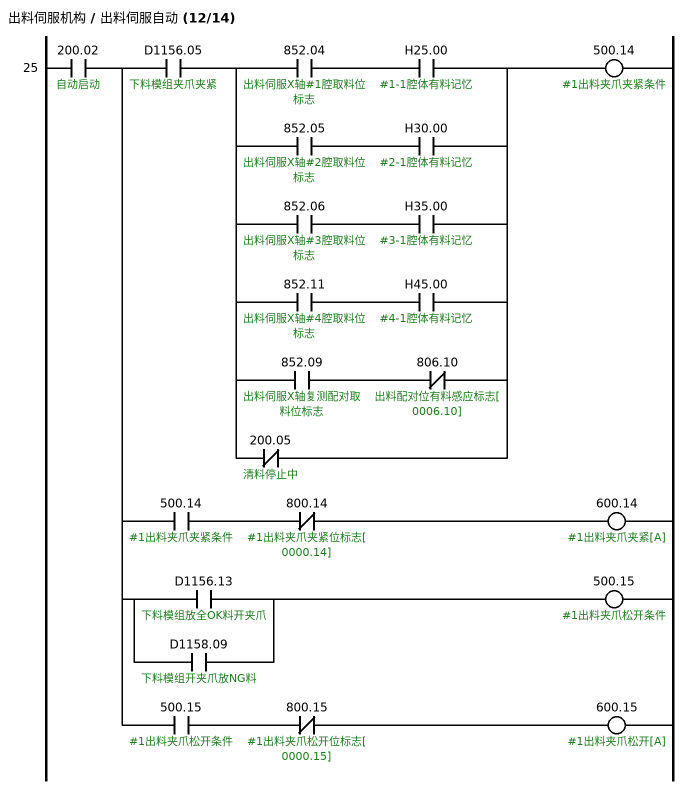
; rung 25
LD 200.02  ; 自动启动
OUT TR0
AND D1156.05  ; 下料模组夹爪夹紧
LD 852.04  ; 出料伺服X轴#1腔取料位标志
AND H25.00  ; #1-1腔体有料记忆
LD 852.05  ; 出料伺服X轴#2腔取料位标志
AND H30.00  ; #2-1腔体有料记忆
ORLD
LD 852.06  ; 出料伺服X轴#3腔取料位标志
AND H35.00  ; #3-1腔体有料记忆
ORLD
LD 852.11  ; 出料伺服X轴#4腔取料位标志
AND H45.00  ; #4-1腔体有料记忆
ORLD
LD 852.09  ; 出料伺服X轴复测配对取料位标志
ANDNOT 806.10  ; 出料配对位有料感应标志[0006.10]
ORLD
ORNOT 200.05  ; 清料停止中
ANDLD
OUT 500.14  ; #1出料夹爪夹紧条件
LD TR0
AND 500.14  ; #1出料夹爪夹紧条件
ANDNOT 800.14  ; #1出料夹爪夹紧位标志[0000.14]
OUT 600.14  ; #1出料夹爪夹紧[A]
LD TR0
LD D1156.13  ; 下料模组放全OK料开夹爪
OR D1158.09  ; 下料模组开夹爪放NG料
ANDLD
OUT 500.15  ; #1出料夹爪松开条件
LD TR0
AND 500.15  ; #1出料夹爪松开条件
ANDNOT 800.15  ; #1出料夹爪松开位标志[0000.15]
OUT 600.15  ; #1出料夹爪松开[A]

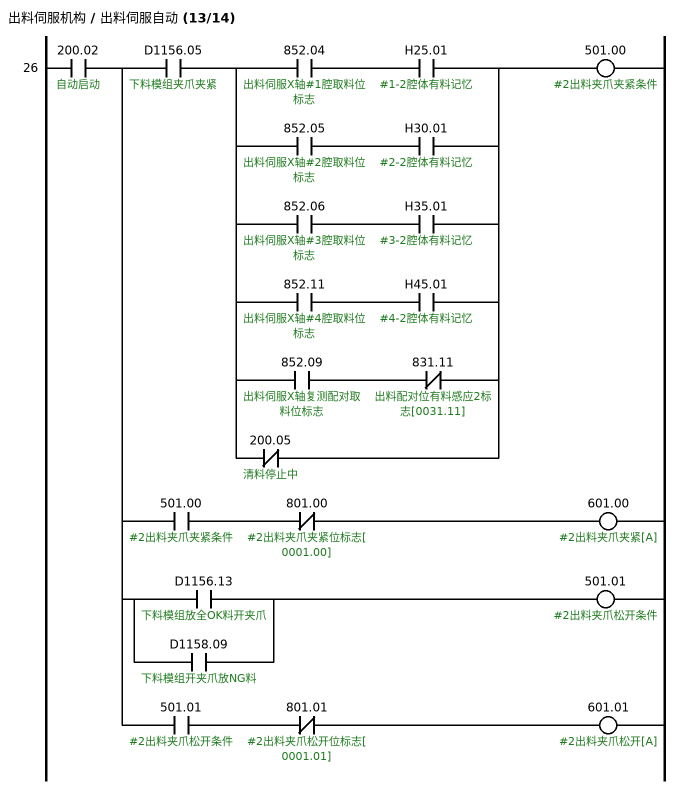
; rung 26
LD 200.02  ; 自动启动
OUT TR0
AND D1156.05  ; 下料模组夹爪夹紧
LD 852.04  ; 出料伺服X轴#1腔取料位标志
AND H25.01  ; #1-2腔体有料记忆
LD 852.05  ; 出料伺服X轴#2腔取料位标志
AND H30.01  ; #2-2腔体有料记忆
ORLD
LD 852.06  ; 出料伺服X轴#3腔取料位标志
AND H35.01  ; #3-2腔体有料记忆
ORLD
LD 852.11  ; 出料伺服X轴#4腔取料位标志
AND H45.01  ; #4-2腔体有料记忆
ORLD
LD 852.09  ; 出料伺服X轴复测配对取料位标志
ANDNOT 831.11  ; 出料配对位有料感应2标志[0031.11]
ORLD
ORNOT 200.05  ; 清料停止中
ANDLD
OUT 501.00  ; #2出料夹爪夹紧条件
LD TR0
AND 501.00  ; #2出料夹爪夹紧条件
ANDNOT 801.00  ; #2出料夹爪夹紧位标志[0001.00]
OUT 601.00  ; #2出料夹爪夹紧[A]
LD TR0
LD D1156.13  ; 下料模组放全OK料开夹爪
OR D1158.09  ; 下料模组开夹爪放NG料
ANDLD
OUT 501.01  ; #2出料夹爪松开条件
LD TR0
AND 501.01  ; #2出料夹爪松开条件
ANDNOT 801.01  ; #2出料夹爪松开位标志[0001.01]
OUT 601.01  ; #2出料夹爪松开[A]

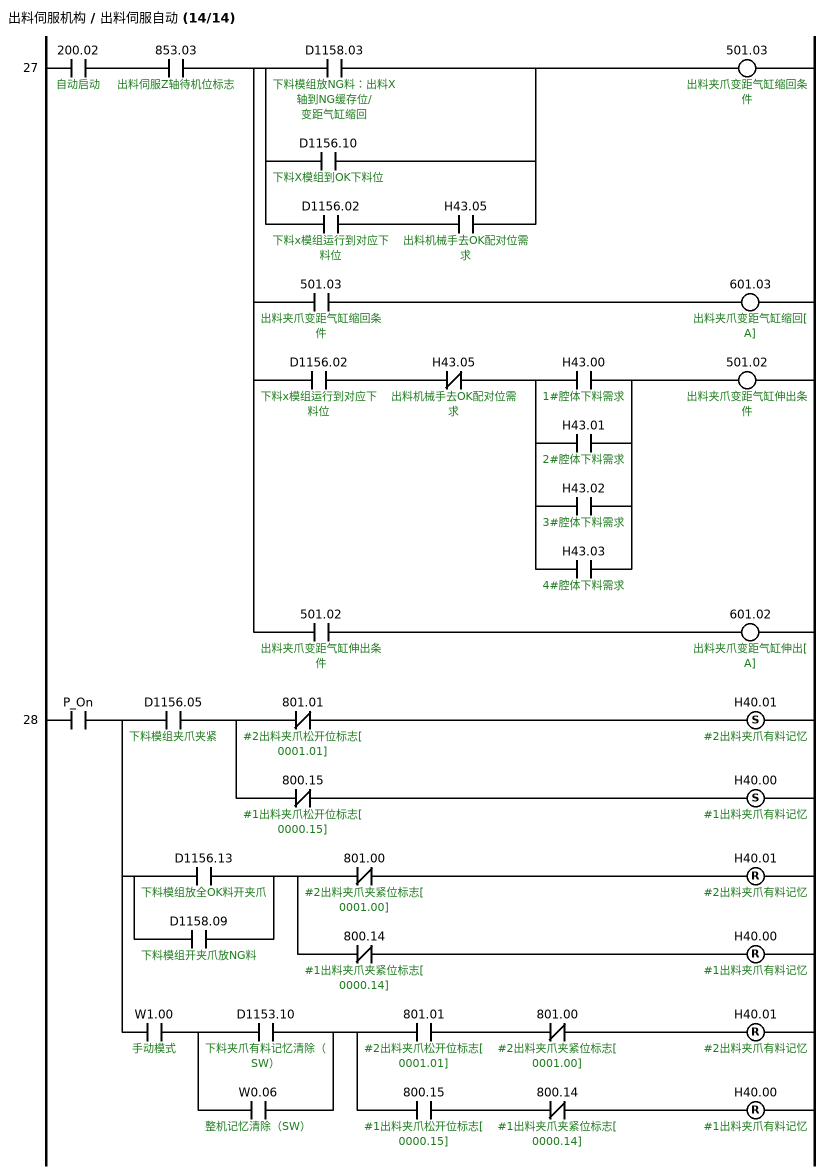
; rung 27
LD 200.02  ; 自动启动
AND 853.03  ; 出料伺服Z轴待机位标志
OUT TR0
LD D1158.03  ; 下料模组放NG料：出料X轴到NG缓存位/变距气缸缩回
OR D1156.10  ; 下料X模组到OK下料位
LD D1156.02  ; 下料x模组运行到对应下料位
AND H43.05  ; 出料机械手去OK配对位需求
ORLD
ANDLD
OUT 501.03  ; 出料夹爪变距气缸缩回条件
LD TR0
AND 501.03  ; 出料夹爪变距气缸缩回条件
OUT 601.03  ; 出料夹爪变距气缸缩回[A]
LD TR0
AND D1156.02  ; 下料x模组运行到对应下料位
ANDNOT H43.05  ; 出料机械手去OK配对位需求
LD H43.00  ; 1#腔体下料需求
OR H43.01  ; 2#腔体下料需求
OR H43.02  ; 3#腔体下料需求
OR H43.03  ; 4#腔体下料需求
ANDLD
OUT 501.02  ; 出料夹爪变距气缸伸出条件
LD TR0
AND 501.02  ; 出料夹爪变距气缸伸出条件
OUT 601.02  ; 出料夹爪变距气缸伸出[A]
; rung 28
LD P_On
OUT TR0
AND D1156.05  ; 下料模组夹爪夹紧
OUT TR1
ANDNOT 801.01  ; #2出料夹爪松开位标志[0001.01]
SET H40.01  ; #2出料夹爪有料记忆
LD TR1
ANDNOT 800.15  ; #1出料夹爪松开位标志[0000.15]
SET H40.00  ; #1出料夹爪有料记忆
LD TR0
LD D1156.13  ; 下料模组放全OK料开夹爪
OR D1158.09  ; 下料模组开夹爪放NG料
ANDLD
OUT TR1
ANDNOT 801.00  ; #2出料夹爪夹紧位标志[0001.00]
RSET H40.01  ; #2出料夹爪有料记忆
LD TR1
ANDNOT 800.14  ; #1出料夹爪夹紧位标志[0000.14]
RSET H40.00  ; #1出料夹爪有料记忆
LD TR0
AND W1.00  ; 手动模式
LD D1153.10  ; 下料夹爪有料记忆清除（SW）
OR W0.06  ; 整机记忆清除（SW）
ANDLD
OUT TR0
AND 801.01  ; #2出料夹爪松开位标志[0001.01]
ANDNOT 801.00  ; #2出料夹爪夹紧位标志[0001.00]
RSET H40.01  ; #2出料夹爪有料记忆
LD TR0
AND 800.15  ; #1出料夹爪松开位标志[0000.15]
ANDNOT 800.14  ; #1出料夹爪夹紧位标志[0000.14]
RSET H40.00  ; #1出料夹爪有料记忆

### Section 工站复位

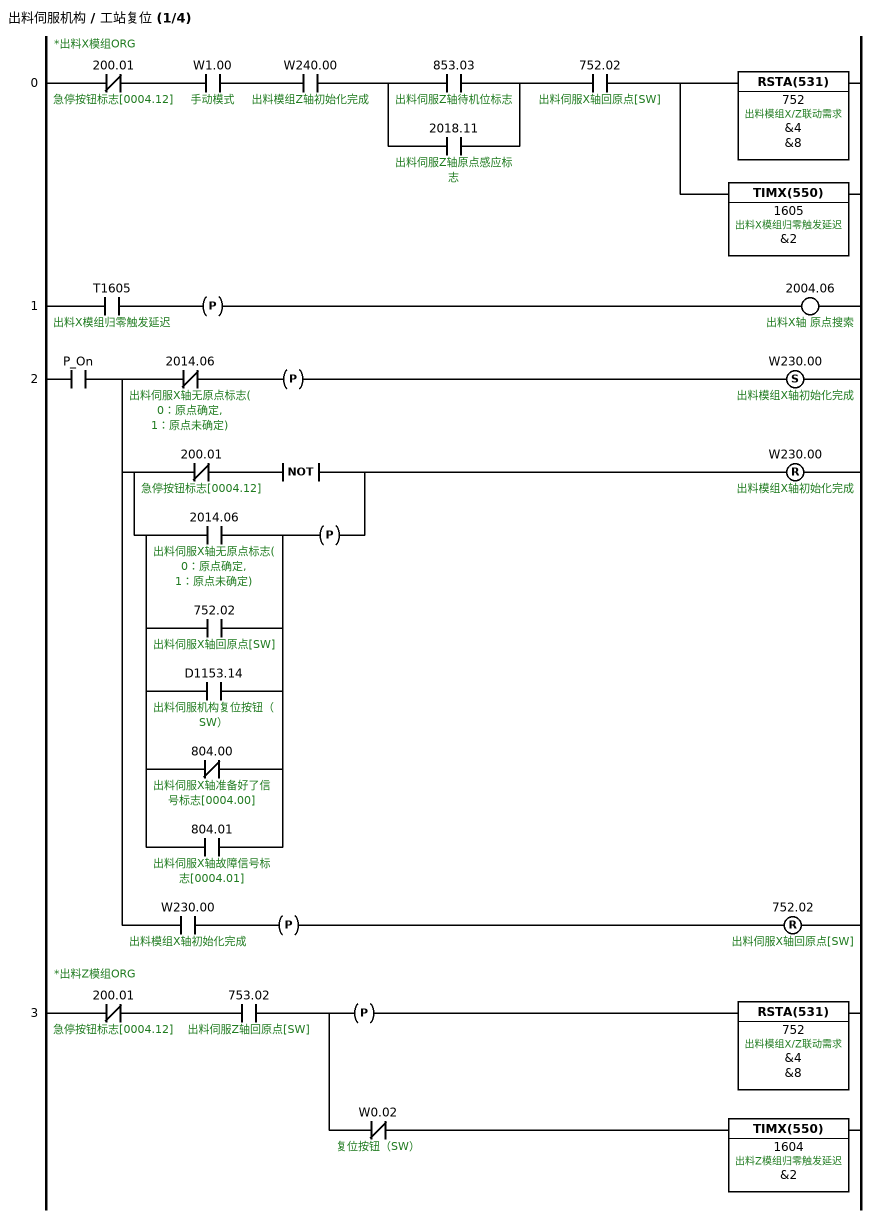
; rung 0: *出料X模组ORG
LDNOT 200.01  ; 急停按钮标志[0004.12]
AND W1.00  ; 手动模式
AND W240.00  ; 出料模组Z轴初始化完成
LD 853.03  ; 出料伺服Z轴待机位标志
OR 2018.11  ; 出料伺服Z轴原点感应标志
ANDLD
AND 752.02  ; 出料伺服X轴回原点[SW]
RSTA(531) 752 &4 &8  ; 出料模组X/Z联动需求
TIMX(550) 1605 &2  ; 出料X模组归零触发延迟
; rung 1
LD T1605  ; 出料X模组归零触发延迟
UP(521)
OUT 2004.06  ; 出料X轴 原点搜索
; rung 2
LD P_On
OUT TR0
ANDNOT 2014.06  ; 出料伺服X轴无原点标志(0：原点确定,1：原点未确定)
UP(521)
SET W230.00  ; 出料模组X轴初始化完成
LD TR0
LDNOT 200.01  ; 急停按钮标志[0004.12]
NOT(520)
LD 2014.06  ; 出料伺服X轴无原点标志(0：原点确定,1：原点未确定)
OR 752.02  ; 出料伺服X轴回原点[SW]
OR D1153.14  ; 出料伺服机构复位按钮（SW）
ORNOT 804.00  ; 出料伺服X轴准备好了信号标志[0004.00]
OR 804.01  ; 出料伺服X轴故障信号标志[0004.01]
UP(521)
ORLD
ANDLD
RSET W230.00  ; 出料模组X轴初始化完成
LD TR0
AND W230.00  ; 出料模组X轴初始化完成
UP(521)
RSET 752.02  ; 出料伺服X轴回原点[SW]
; rung 3: *出料Z模组ORG
LDNOT 200.01  ; 急停按钮标志[0004.12]
AND 753.02  ; 出料伺服Z轴回原点[SW]
OUT TR0
UP(521)
RSTA(531) 752 &4 &8  ; 出料模组X/Z联动需求
LD TR0
ANDNOT W0.02  ; 复位按钮（SW）
TIMX(550) 1604 &2  ; 出料Z模组归零触发延迟

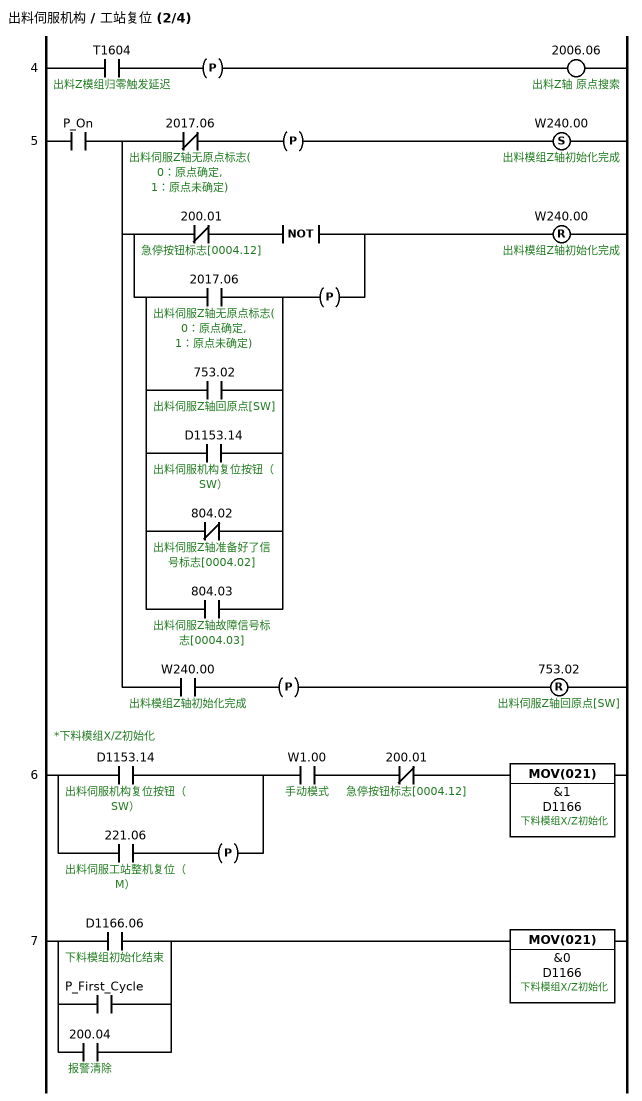
; rung 4
LD T1604  ; 出料Z模组归零触发延迟
UP(521)
OUT 2006.06  ; 出料Z轴 原点搜索
; rung 5
LD P_On
OUT TR0
ANDNOT 2017.06  ; 出料伺服Z轴无原点标志(0：原点确定,1：原点未确定)
UP(521)
SET W240.00  ; 出料模组Z轴初始化完成
LD TR0
LDNOT 200.01  ; 急停按钮标志[0004.12]
NOT(520)
LD 2017.06  ; 出料伺服Z轴无原点标志(0：原点确定,1：原点未确定)
OR 753.02  ; 出料伺服Z轴回原点[SW]
OR D1153.14  ; 出料伺服机构复位按钮（SW）
ORNOT 804.02  ; 出料伺服Z轴准备好了信号标志[0004.02]
OR 804.03  ; 出料伺服Z轴故障信号标志[0004.03]
UP(521)
ORLD
ANDLD
RSET W240.00  ; 出料模组Z轴初始化完成
LD TR0
AND W240.00  ; 出料模组Z轴初始化完成
UP(521)
RSET 753.02  ; 出料伺服Z轴回原点[SW]
; rung 6: *下料模组X/Z初始化
LD D1153.14  ; 出料伺服机构复位按钮（SW）
LD 221.06  ; 出料伺服工站整机复位（M）
UP(521)
ORLD
AND W1.00  ; 手动模式
ANDNOT 200.01  ; 急停按钮标志[0004.12]
MOV(021) &1 D1166  ; 下料模组X/Z初始化
; rung 7
LD D1166.06  ; 下料模组初始化结束
OR P_First_Cycle
OR 200.04  ; 报警清除
MOV(021) &0 D1166  ; 下料模组X/Z初始化

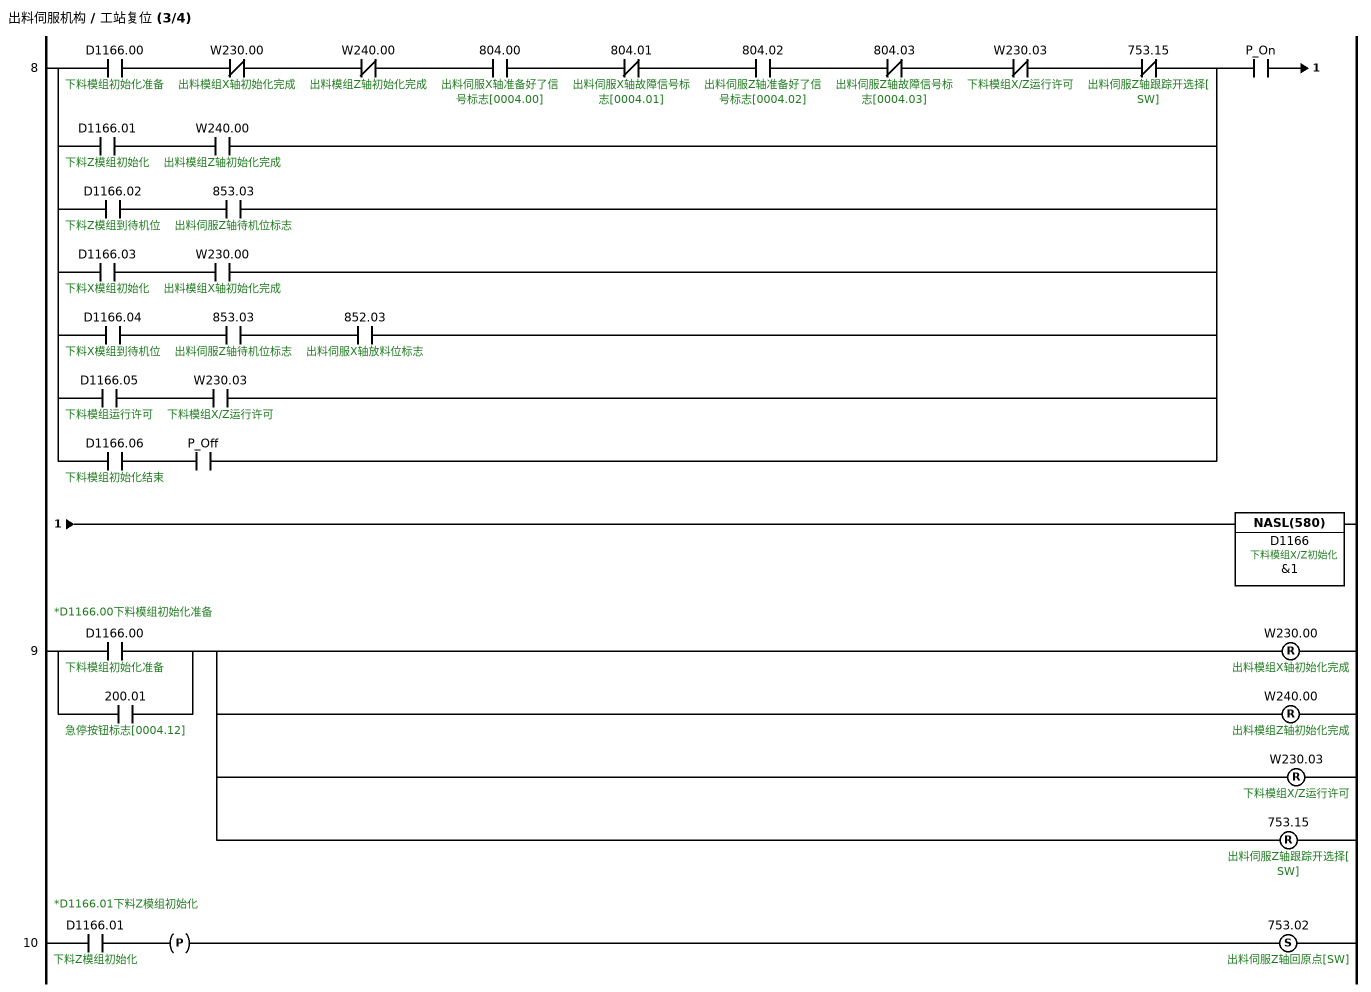
; rung 8
LD D1166.00  ; 下料模组初始化准备
ANDNOT W230.00  ; 出料模组X轴初始化完成
ANDNOT W240.00  ; 出料模组Z轴初始化完成
AND 804.00  ; 出料伺服X轴准备好了信号标志[0004.00]
ANDNOT 804.01  ; 出料伺服X轴故障信号标志[0004.01]
AND 804.02  ; 出料伺服Z轴准备好了信号标志[0004.02]
ANDNOT 804.03  ; 出料伺服Z轴故障信号标志[0004.03]
ANDNOT W230.03  ; 下料模组X/Z运行许可
ANDNOT 753.15  ; 出料伺服Z轴跟踪开选择[SW]
LD D1166.01  ; 下料Z模组初始化
AND W240.00  ; 出料模组Z轴初始化完成
ORLD
LD D1166.02  ; 下料Z模组到待机位
AND 853.03  ; 出料伺服Z轴待机位标志
ORLD
LD D1166.03  ; 下料X模组初始化
AND W230.00  ; 出料模组X轴初始化完成
ORLD
LD D1166.04  ; 下料X模组到待机位
AND 853.03  ; 出料伺服Z轴待机位标志
AND 852.03  ; 出料伺服X轴放料位标志
ORLD
LD D1166.05  ; 下料模组运行许可
AND W230.03  ; 下料模组X/Z运行许可
ORLD
LD D1166.06  ; 下料模组初始化结束
AND P_Off
ORLD
AND P_On
NASL(580) D1166 &1  ; 下料模组X/Z初始化
; rung 9: *D1166.00下料模组初始化准备
LD D1166.00  ; 下料模组初始化准备
OR 200.01  ; 急停按钮标志[0004.12]
RSET W230.00  ; 出料模组X轴初始化完成
RSET W240.00  ; 出料模组Z轴初始化完成
RSET W230.03  ; 下料模组X/Z运行许可
RSET 753.15  ; 出料伺服Z轴跟踪开选择[SW]
; rung 10: *D1166.01下料Z模组初始化
LD D1166.01  ; 下料Z模组初始化
UP(521)
SET 753.02  ; 出料伺服Z轴回原点[SW]

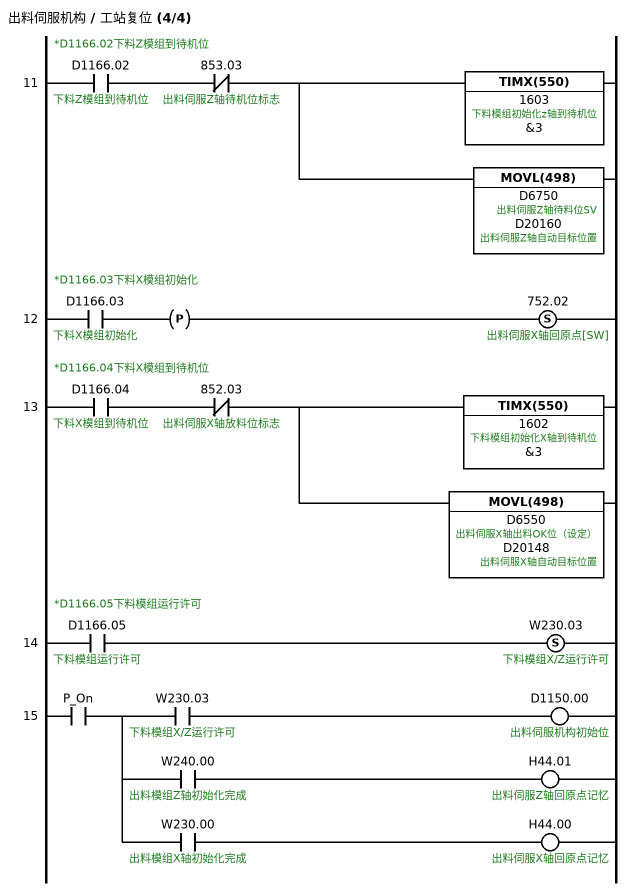
; rung 11: *D1166.02下料Z模组到待机位
LD D1166.02  ; 下料Z模组到待机位
ANDNOT 853.03  ; 出料伺服Z轴待机位标志
TIMX(550) 1603 &3  ; 下料模组初始化z轴到待机位
MOVL(498) D6750 D20160  ; 出料伺服Z轴待料位SV, 出料伺服Z轴自动目标位置
; rung 12: *D1166.03下料X模组初始化
LD D1166.03  ; 下料X模组初始化
UP(521)
SET 752.02  ; 出料伺服X轴回原点[SW]
; rung 13: *D1166.04下料X模组到待机位
LD D1166.04  ; 下料X模组到待机位
ANDNOT 852.03  ; 出料伺服X轴放料位标志
TIMX(550) 1602 &3  ; 下料模组初始化X轴到待机位
MOVL(498) D6550 D20148  ; 出料伺服X轴出料OK位（设定）, 出料伺服X轴自动目标位置
; rung 14: *D1166.05下料模组运行许可
LD D1166.05  ; 下料模组运行许可
SET W230.03  ; 下料模组X/Z运行许可
; rung 15
LD P_On
OUT TR0
AND W230.03  ; 下料模组X/Z运行许可
OUT D1150.00  ; 出料伺服机构初始位
LD TR0
AND W240.00  ; 出料模组Z轴初始化完成
OUT H44.01  ; 出料伺服Z轴回原点记忆
LD TR0
AND W230.00  ; 出料模组X轴初始化完成
OUT H44.00  ; 出料伺服X轴回原点记忆

### Section 指示灯

